LIN {X 0,Y 204.772,Z 618.344,A -85,B 0,C 180,E1 -29638.617,E2 -29638.617} C_VEL
LIN {X 0,Y 211.612,Z 616.813,A -85,B 0,C 180,E1 -29641.984,E2 -29641.984} C_VEL
LIN {X 0,Y 215.146,Z 615.633,A -85,B 0,C 180,E1 -29643.61,E2 -29643.61} C_VEL
LIN {X 0,Y 223.244,Z 612.344,A -85,B 0,C 180,E1 -29646.599,E2 -29646.599} C_VEL
LIN {X 0,Y 232.156,Z 607.768,A -85,B 0,C 180,E1 -29649.321,E2 -29649.321} C_VEL
LIN {X 0,Y 241.752,Z 601.799,A -85,B 0,C 180,E1 -29651.794,E2 -29651.794} C_VEL
LIN {X 0,Y 251.918,Z 594.305,A -85,B 0,C 180,E1 -29654.041,E2 -29654.041} C_VEL
LIN {X 0,Y 261.51,Z 586.109,A -85,B 0,C 180,E1 -29655.824,E2 -29655.824} C_VEL
LIN {X 0,Y 271.184,Z 576.576,A -85,B 0,C 180,E1 -29657.407,E2 -29657.407} C_VEL
LIN {X 0,Y 279.896,Z 566.683,A -85,B 0,C 180,E1 -29658.66,E2 -29658.66} C_VEL
LIN {X 0,Y 288.902,Z 554.834,A -85,B 0,C 180,E1 -29659.797,E2 -29659.797} C_VEL
LIN {X 0,Y 297.375,Z 541.679,A -85,B 0,C 180,E1 -29660.75,E2 -29660.75} C_VEL
LIN {X 0,Y 300.334,Z 536.479,A -85,B 0,C 180,E1 -29661.053,E2 -29661.053} C_VEL
LIN {X 0,Y 300.286,Z 536.529,A -85,B 0,C 180,E1 -29661.393,E2 -29661.393} C_VEL
LIN {X 0,Y 292.719,Z 549.042,A -85,B 0,C 180,E1 -29662.328,E2 -29662.328} C_VEL
LIN {X 0,Y 284.753,Z 560.194,A -85,B 0,C 180,E1 -29663.38,E2 -29663.38} C_VEL
LIN {X 0,Y 275.713,Z 571.006,A -85,B 0,C 180,E1 -29664.684,E2 -29664.684} C_VEL
LIN {X 0,Y 266.952,Z 580.103,A -85,B 0,C 180,E1 -29666.112,E2 -29666.112} C_VEL
LIN {X 0,Y 256.846,Z 589.123,A -85,B 0,C 180,E1 -29667.977,E2 -29667.977} C_VEL
LIN {X 0,Y 246.497,Z 596.964,A -85,B 0,C 180,E1 -29670.18,E2 -29670.18} C_VEL
LIN {X 0,Y 236.497,Z 603.258,A -85,B 0,C 180,E1 -29672.696,E2 -29672.696} C_VEL
LIN {X 0,Y 227.293,Z 607.968,A -85,B 0,C 180,E1 -29675.416,E2 -29675.416} C_VEL
LIN {X 0,Y 218.078,Z 611.557,A -85,B 0,C 180,E1 -29678.672,E2 -29678.672} C_VEL
LIN {X 0,Y 212.957,Z 613.013,A -85,B 0,C 180,E1 -29680.797,E2 -29680.797} C_VEL
LIN {X 0,Y 205.913,Z 614.151,A -85,B 0,C 180,E1 -29684.209,E2 -29684.209} C_VEL
LIN {X 0,Y 199.91,Z 614.063,A -85,B 0,C 180,E1 -29687.864,E2 -29687.864} C_VEL
LIN {X 0,Y 195.099,Z 612.779,A -85,B 0,C 180,E1 -29691.743,E2 -29691.743} C_VEL
LIN {X 0,Y 191.462,Z 610.312,A -85,B 0,C 180,E1 -29695.804,E2 -29695.804} C_VEL
LIN {X 0,Y 188.992,Z 606.632,A -85,B 0,C 180,E1 -29700,E2 -29700} C_VEL
LIN {X 0,Y 187.534,Z 601.624,A -85,B 0,C 180,E1 -29704.284,E2 -29704.284} C_VEL
LIN {X 0,Y 187.042,Z 595.113,A -85,B 0,C 180,E1 -29708.615,E2 -29708.615} C_VEL
LIN {X 0,Y 187.164,Z 587.88,A -85,B 0,C 180,E1 -29712.427,E2 -29712.427} C_VEL
LIN {X 0,Y 187.494,Z 580.247,A -85,B 0,C 180,E1 -29715.715,E2 -29715.715} C_VEL
LIN {X 0,Y 187.907,Z 570.867,A -85,B 0,C 180,E1 -29719.036,E2 -29719.036} C_VEL
LIN {X 0,Y 188.535,Z 560.39,A -85,B 0,C 180,E1 -29722.096,E2 -29722.096} C_VEL
LIN {X 0,Y 189.361,Z 548.884,A -85,B 0,C 180,E1 -29724.883,E2 -29724.883} C_VEL
LIN {X 0,Y 190.461,Z 535.611,A -85,B 0,C 180,E1 -29727.516,E2 -29727.516} C_VEL
LIN {X 0,Y 191.581,Z 521.627,A -85,B 0,C 180,E1 -29729.727,E2 -29729.727} C_VEL
LIN {X 0,Y 192.62,Z 507.163,A -85,B 0,C 180,E1 -29731.516,E2 -29731.516} C_VEL
LIN {X 0,Y 193.716,Z 492.08,A -85,B 0,C 180,E1 -29732.933,E2 -29732.933} C_VEL
LIN {X 0,Y 194.887,Z 470.161,A -85,B 0,C 180,E1 -29734.369,E2 -29734.369} C_VEL
LIN {X 0,Y 198.573,Z 392.946,A -85,B 0,C 180,E1 -29738.995,E2 -29738.995} C_VEL
LIN {X 0,Y 195.924,Z 362.092,A -85,B 0,C 180,E1 -29740.947,E2 -29740.947} C_VEL
LIN {X 0,Y 192.683,Z 347.917,A -85,B 0,C 180,E1 -29742.011,E2 -29742.011} C_VEL
LIN {X 0,Y 189.766,Z 333.395,A -85,B 0,C 180,E1 -29746.279,E2 -29746.279} C_VEL
LIN {X 0,Y 189.689,Z 333.409,A -85,B 0,C 180,E1 -29751.11,E2 -29751.11} C_VEL
LIN {X 0,Y 189.64,Z 333.393,A -85,B 0,C 180,E1 -29756.35,E2 -29756.35} C_VEL
LIN {X 0,Y 189.682,Z 333.399,A -85,B 0,C 180,E1 -29757.777,E2 -29757.777} C_VEL
LIN {X 0,Y 190.707,Z 336.248,A -85,B 0,C 180,E1 -29758.187,E2 -29758.187} C_VEL
LIN {X 0,Y 192.446,Z 338.584,A -85,B 0,C 180,E1 -29758.713,E2 -29758.713} C_VEL
LIN {X 0,Y 201.749,Z 354.151,A -85,B 0,C 180,E1 -29761.457,E2 -29761.457} C_VEL
LIN {X 0,Y 210.076,Z 370.517,A -85,B 0,C 180,E1 -29763.742,E2 -29763.742} C_VEL
LIN {X 0,Y 214.586,Z 381.294,A -85,B 0,C 180,E1 -29764.958,E2 -29764.958} C_VEL
LIN {X 0,Y 210.894,Z 456.713,A -85,B 0,C 180,E1 -29767.348,E2 -29767.348} C_VEL
LIN {X 0,Y 209.707,Z 470.555,A -85,B 0,C 180,E1 -29768.117,E2 -29768.117} C_VEL
LIN {X 0,Y 207.974,Z 484.658,A -85,B 0,C 180,E1 -29769.286,E2 -29769.286} C_VEL
LIN {X 0,Y 205.708,Z 498.601,A -85,B 0,C 180,E1 -29770.864,E2 -29770.864} C_VEL
LIN {X 0,Y 202.935,Z 511.157,A -85,B 0,C 180,E1 -29772.676,E2 -29772.676} C_VEL
LIN {X 0,Y 200.212,Z 522.577,A -85,B 0,C 180,E1 -29774.783,E2 -29774.783} C_VEL
LIN {X 0,Y 198.207,Z 531.077,A -85,B 0,C 180,E1 -29776.716,E2 -29776.716} C_VEL
LIN {X 0,Y 195.137,Z 541.849,A -85,B 0,C 180,E1 -29779.656,E2 -29779.656} C_VEL
LIN {X 0,Y 192.712,Z 550.717,A -85,B 0,C 180,E1 -29782.686,E2 -29782.686} C_VEL
LIN {X 0,Y 190.577,Z 558.125,A -85,B 0,C 180,E1 -29785.779,E2 -29785.779} C_VEL
LIN {X 0,Y 189.135,Z 564.829,A -85,B 0,C 180,E1 -29789.266,E2 -29789.266} C_VEL
LIN {X 0,Y 187.809,Z 570.83,A -85,B 0,C 180,E1 -29793.202,E2 -29793.202} C_VEL
LIN {X 0,Y 186.836,Z 575.79,A -85,B 0,C 180,E1 -29797.534,E2 -29797.534} C_VEL
LIN {X 0,Y 186.652,Z 578.504,A -85,B 0,C 180,E1 -29800.809,E2 -29800.809} C_VEL
LIN {X 0,Y 186.756,Z 579.872,A -85,B 0,C 180,E1 -29802.999,E2 -29802.999} C_VEL
LIN {X 0,Y 187.345,Z 581.595,A -85,B 0,C 180,E1 -29807.398,E2 -29807.398} C_VEL
LIN {X 0,Y 188.986,Z 581.937,A -85,B 0,C 180,E1 -29812.092,E2 -29812.092} C_VEL
LIN {X 0,Y 191.122,Z 580.952,A -85,B 0,C 180,E1 -29816.084,E2 -29816.084} C_VEL
LIN {X 0,Y 194.361,Z 578.551,A -85,B 0,C 180,E1 -29820.294,E2 -29820.294} C_VEL
LIN {X 0,Y 198.436,Z 574.642,A -85,B 0,C 180,E1 -29824.38,E2 -29824.38} C_VEL
LIN {X 0,Y 203.477,Z 569.082,A -85,B 0,C 180,E1 -29828.282,E2 -29828.282} C_VEL
LIN {X 0,Y 208.517,Z 562.735,A -85,B 0,C 180,E1 -29831.555,E2 -29831.555} C_VEL
LIN {X 0,Y 214.19,Z 554.762,A -85,B 0,C 180,E1 -29834.668,E2 -29834.668} C_VEL
LIN {X 0,Y 219.487,Z 546.356,A -85,B 0,C 180,E1 -29837.215,E2 -29837.215} C_VEL
LIN {X 0,Y 225.215,Z 536.161,A -85,B 0,C 180,E1 -29839.631,E2 -29839.631} C_VEL
LIN {X 0,Y 230.243,Z 525.826,A -85,B 0,C 180,E1 -29841.562,E2 -29841.562} C_VEL
LIN {X 0,Y 234.956,Z 514.4,A -85,B 0,C 180,E1 -29843.274,E2 -29843.274} C_VEL
LIN {X 0,Y 239.109,Z 502.35,A -85,B 0,C 180,E1 -29844.698,E2 -29844.698} C_VEL
LIN {X 0,Y 242.65,Z 489.425,A -85,B 0,C 180,E1 -29845.896,E2 -29845.896} C_VEL
LIN {X 0,Y 245.689,Z 475.198,A -85,B 0,C 180,E1 -29846.854,E2 -29846.854} C_VEL
LIN {X 0,Y 247.681,Z 461.5,A -85,B 0,C 180,E1 -29847.513,E2 -29847.513} C_VEL
LIN {X 0,Y 249.394,Z 440.592,A -85,B 0,C 180,E1 -29848.12,E2 -29848.12} C_VEL
LIN {X 0,Y 251.105,Z 416.237,A -85,B 0,C 180,E1 -29848.742,E2 -29848.742} C_VEL
LIN {X 0,Y 244.75,Z 404.193,A -85,B 0,C 180,E1 -29851.331,E2 -29851.331} C_VEL
LIN {X 0,Y 239.319,Z 395.049,A -85,B 0,C 180,E1 -29853.74,E2 -29853.74} C_VEL
LIN {X 0,Y 234.137,Z 386.937,A -85,B 0,C 180,E1 -29856.29,E2 -29856.29} C_VEL
LIN {X 0,Y 229.497,Z 380.171,A -85,B 0,C 180,E1 -29858.838,E2 -29858.838} C_VEL
LIN {X 0,Y 226.579,Z 376.111,A -85,B 0,C 180,E1 -29860.605,E2 -29860.605} C_VEL
LIN {X 0,Y 223.563,Z 371.946,A -85,B 0,C 180,E1 -29862.612,E2 -29862.612} C_VEL
LIN {X 0,Y 220.384,Z 367.707,A -85,B 0,C 180,E1 -29864.976,E2 -29864.976} C_VEL
LIN {X 0,Y 217.707,Z 364.529,A -85,B 0,C 180,E1 -29867.206,E2 -29867.206} C_VEL
LIN {X 0,Y 216.596,Z 362.722,A -85,B 0,C 180,E1 -29868.28,E2 -29868.28} C_VEL
LIN {X 0,Y 214.036,Z 360.136,A -85,B 0,C 180,E1 -29870.924,E2 -29870.924} C_VEL
LIN {X 0,Y 212.711,Z 357.426,A -85,B 0,C 180,E1 -29872.728,E2 -29872.728} C_VEL
LIN {X 0,Y 209.928,Z 355.08,A -85,B 0,C 180,E1 -29877.071,E2 -29877.071} C_VEL
LIN {X 0,Y 208.728,Z 352.105,A -85,B 0,C 180,E1 -29880.602,E2 -29880.602} C_VEL
LIN {X 0,Y 208.657,Z 351.751,A -85,B 0,C 180,E1 -29880.963,E2 -29880.963} C_VEL
LIN {X 0,Y 208.195,Z 351.882,A -85,B 0,C 180,E1 -29888.464,E2 -29888.464} C_VEL
LIN {X 0,Y 208.512,Z 352.77,A -85,B 0,C 180,E1 -29890.219,E2 -29890.219} C_VEL
LIN {X 0,Y 210.498,Z 356.559,A -85,B 0,C 180,E1 -29895.439,E2 -29895.439} C_VEL
LIN {X 0,Y 213.777,Z 361.036,A -85,B 0,C 180,E1 -29900.192,E2 -29900.192} C_VEL
LIN {X 0,Y 218.035,Z 367.529,A -85,B 0,C 180,E1 -29904.59,E2 -29904.59} C_VEL
LIN {X 0,Y 222.816,Z 375.197,A -85,B 0,C 180,E1 -29908.454,E2 -29908.454} C_VEL
LIN {X 0,Y 226.433,Z 381.12,A -85,B 0,C 180,E1 -29910.933,E2 -29910.933} C_VEL
LIN {X 0,Y 230.081,Z 387.521,A -85,B 0,C 180,E1 -29913.184,E2 -29913.184} C_VEL
LIN {X 0,Y 234.473,Z 395.589,A -85,B 0,C 180,E1 -29915.629,E2 -29915.629} C_VEL
LIN {X 0,Y 239.381,Z 405.545,A -85,B 0,C 180,E1 -29918.107,E2 -29918.107} C_VEL
LIN {X 0,Y 244.569,Z 417.022,A -85,B 0,C 180,E1 -29920.506,E2 -29920.506} C_VEL
LIN {X 0,Y 249.126,Z 428.767,A -85,B 0,C 180,E1 -29922.503,E2 -29922.503} C_VEL
LIN {X 0,Y 249.583,Z 430.837,A -85,B 0,C 180,E1 -29922.735,E2 -29922.735} C_VEL
LIN {X 0,Y 249.848,Z 436.032,A -85,B 0,C 180,E1 -29923.052,E2 -29923.052} C_VEL
LIN {X 0,Y 246.628,Z 477.617,A -85,B 0,C 180,E1 -29924.114,E2 -29924.114} C_VEL
LIN {X 0,Y 244.414,Z 491.839,A -85,B 0,C 180,E1 -29924.684,E2 -29924.684} C_VEL
LIN {X 0,Y 241.258,Z 506.122,A -85,B 0,C 180,E1 -29925.546,E2 -29925.546} C_VEL
LIN {X 0,Y 237.076,Z 519.77,A -85,B 0,C 180,E1 -29926.62,E2 -29926.62} C_VEL
LIN {X 0,Y 232.475,Z 532.04,A -85,B 0,C 180,E1 -29927.909,E2 -29927.909} C_VEL
LIN {X 0,Y 227.643,Z 543.281,A -85,B 0,C 180,E1 -29929.465,E2 -29929.465} C_VEL
LIN {X 0,Y 222.898,Z 552.692,A -85,B 0,C 180,E1 -29931.068,E2 -29931.068} C_VEL
LIN {X 0,Y 219.363,Z 559.338,A -85,B 0,C 180,E1 -29932.452,E2 -29932.452} C_VEL
LIN {X 0,Y 216.541,Z 563.417,A -85,B 0,C 180,E1 -29933.297,E2 -29933.297} C_VEL
LIN {X 0,Y 210.353,Z 569.669,A -85,B 0,C 180,E1 -29934.529,E2 -29934.529} C_VEL
LIN {X 0,Y 204.048,Z 575.426,A -85,B 0,C 180,E1 -29935.933,E2 -29935.933} C_VEL
LIN {X 0,Y 201.095,Z 578.671,A -85,B 0,C 180,E1 -29937.048,E2 -29937.048} C_VEL
LIN {X 0,Y 195.998,Z 585.222,A -85,B 0,C 180,E1 -29939.985,E2 -29939.985} C_VEL
LIN {X 0,Y 190.604,Z 591.683,A -85,B 0,C 180,E1 -29943.839,E2 -29943.839} C_VEL
LIN {X 0,Y 186.379,Z 596.566,A -85,B 0,C 180,E1 -29947.931,E2 -29947.931} C_VEL
LIN {X 0,Y 183.063,Z 600.003,A -85,B 0,C 180,E1 -29952.182,E2 -29952.182} C_VEL
LIN {X 0,Y 180.819,Z 602.091,A -85,B 0,C 180,E1 -29956.566,E2 -29956.566} C_VEL
LIN {X 0,Y 179.627,Z 602.882,A -85,B 0,C 180,E1 -29961.032,E2 -29961.032} C_VEL
LIN {X 0,Y 179.587,Z 602.391,A -85,B 0,C 180,E1 -29965.532,E2 -29965.532} C_VEL
LIN {X 0,Y 180.477,Z 600.589,A -85,B 0,C 180,E1 -29970.005,E2 -29970.005} C_VEL
LIN {X 0,Y 181.269,Z 598.812,A -85,B 0,C 180,E1 -29972.774,E2 -29972.774} C_VEL
LIN {X 0,Y 180.846,Z 604.623,A -85,B 0,C 180,E1 -29976.678,E2 -29976.678} C_VEL
LIN {X 0,Y 181.12,Z 609.795,A -85,B 0,C 180,E1 -29981.154,E2 -29981.154} C_VEL
LIN {X 0,Y 182.865,Z 613.729,A -85,B 0,C 180,E1 -29985.558,E2 -29985.558} C_VEL
LIN {X 0,Y 185.901,Z 616.471,A -85,B 0,C 180,E1 -29989.828,E2 -29989.828} C_VEL
LIN {X 0,Y 190.04,Z 618.055,A -85,B 0,C 180,E1 -29993.924,E2 -29993.924} C_VEL
LIN {X 0,Y 195.425,Z 618.533,A -85,B 0,C 180,E1 -29997.777,E2 -29997.777} C_VEL
LIN {X 0,Y 202.009,Z 617.902,A -85,B 0,C 180,E1 -30001.345,E2 -30001.345} C_VEL
LIN {X 0,Y 209.302,Z 616.159,A -85,B 0,C 180,E1 -30004.68,E2 -30004.68} C_VEL
LIN {X 0,Y 217.637,Z 613.252,A -85,B 0,C 180,E1 -30007.703,E2 -30007.703} C_VEL
LIN {X 0,Y 226.788,Z 609.104,A -85,B 0,C 180,E1 -30010.441,E2 -30010.441} C_VEL
LIN {X 0,Y 236.63,Z 603.619,A -85,B 0,C 180,E1 -30012.913,E2 -30012.913} C_VEL
LIN {X 0,Y 247.027,Z 596.699,A -85,B 0,C 180,E1 -30015.148,E2 -30015.148} C_VEL
LIN {X 0,Y 255.69,Z 590.016,A -85,B 0,C 180,E1 -30016.73,E2 -30016.73} C_VEL
LIN {X 0,Y 265.231,Z 581.579,A -85,B 0,C 180,E1 -30018.254,E2 -30018.254} C_VEL
LIN {X 0,Y 274.014,Z 572.664,A -85,B 0,C 180,E1 -30019.511,E2 -30019.511} C_VEL
LIN {X 0,Y 283.084,Z 562.119,A -85,B 0,C 180,E1 -30020.649,E2 -30020.649} C_VEL
LIN {X 0,Y 287.744,Z 556.036,A -85,B 0,C 180,E1 -30021.17,E2 -30021.17} C_VEL
LIN {X 0,Y 287.155,Z 556.784,A -85,B 0,C 180,E1 -30021.519,E2 -30021.519} C_VEL
LIN {X 0,Y 277.723,Z 568.304,A -85,B 0,C 180,E1 -30022.749,E2 -30022.749} C_VEL
LIN {X 0,Y 268.759,Z 577.696,A -85,B 0,C 180,E1 -30024.037,E2 -30024.037} C_VEL
LIN {X 0,Y 258.34,Z 587.079,A -85,B 0,C 180,E1 -30025.764,E2 -30025.764} C_VEL
LIN {X 0,Y 248.476,Z 594.599,A -85,B 0,C 180,E1 -30027.615,E2 -30027.615} C_VEL
LIN {X 0,Y 240.38,Z 599.92,A -85,B 0,C 180,E1 -30029.341,E2 -30029.341} C_VEL
LIN {X 0,Y 230.458,Z 605.455,A -85,B 0,C 180,E1 -30031.82,E2 -30031.82} C_VEL
LIN {X 0,Y 223.097,Z 608.777,A -85,B 0,C 180,E1 -30033.925,E2 -30033.925} C_VEL
LIN {X 0,Y 214.2,Z 611.931,A -85,B 0,C 180,E1 -30036.896,E2 -30036.896} C_VEL
LIN {X 0,Y 206.151,Z 613.805,A -85,B 0,C 180,E1 -30040.137,E2 -30040.137} C_VEL
LIN {X 0,Y 198.965,Z 614.461,A -85,B 0,C 180,E1 -30043.642,E2 -30043.642} C_VEL
LIN {X 0,Y 192.894,Z 613.909,A -85,B 0,C 180,E1 -30047.416,E2 -30047.416} C_VEL
LIN {X 0,Y 188.015,Z 612.183,A -85,B 0,C 180,E1 -30051.43,E2 -30051.43} C_VEL
LIN {X 0,Y 184.356,Z 609.288,A -85,B 0,C 180,E1 -30055.642,E2 -30055.642} C_VEL
LIN {X 0,Y 181.653,Z 604.435,A -85,B 0,C 180,E1 -30060.679,E2 -30060.679} C_VEL
LIN {X 0,Y 180.539,Z 599.69,A -85,B 0,C 180,E1 -30064.45,E2 -30064.45} C_VEL
LIN {X 0,Y 180.131,Z 592.661,A -85,B 0,C 180,E1 -30068.948,E2 -30068.948} C_VEL
LIN {X 0,Y 180.336,Z 584.928,A -85,B 0,C 180,E1 -30072.905,E2 -30072.905} C_VEL
LIN {X 0,Y 180.656,Z 576.677,A -85,B 0,C 180,E1 -30076.326,E2 -30076.326} C_VEL
LIN {X 0,Y 181.143,Z 566.602,A -85,B 0,C 180,E1 -30079.776,E2 -30079.776} C_VEL
LIN {X 0,Y 181.822,Z 555.241,A -85,B 0,C 180,E1 -30082.958,E2 -30082.958} C_VEL
LIN {X 0,Y 182.745,Z 542.615,A -85,B 0,C 180,E1 -30085.849,E2 -30085.849} C_VEL
LIN {X 0,Y 183.856,Z 529.323,A -85,B 0,C 180,E1 -30088.332,E2 -30088.332} C_VEL
LIN {X 0,Y 185.016,Z 515.203,A -85,B 0,C 180,E1 -30090.422,E2 -30090.422} C_VEL
LIN {X 0,Y 186.085,Z 500.378,A -85,B 0,C 180,E1 -30092.119,E2 -30092.119} C_VEL
LIN {X 0,Y 187.091,Z 484.465,A -85,B 0,C 180,E1 -30093.439,E2 -30093.439} C_VEL
LIN {X 0,Y 191.458,Z 393.062,A -85,B 0,C 180,E1 -30099.202,E2 -30099.202} C_VEL
LIN {X 0,Y 188.969,Z 363.416,A -85,B 0,C 180,E1 -30101.142,E2 -30101.142} C_VEL
LIN {X 0,Y 185.562,Z 348.298,A -85,B 0,C 180,E1 -30102.257,E2 -30102.257} C_VEL
LIN {X 0,Y 182.722,Z 334.274,A -85,B 0,C 180,E1 -30106.511,E2 -30106.511} C_VEL
LIN {X 0,Y 182.589,Z 334.299,A -85,B 0,C 180,E1 -30112.13,E2 -30112.13} C_VEL
LIN {X 0,Y 182.589,Z 334.283,A -85,B 0,C 180,E1 -30116,E2 -30116} C_VEL
LIN {X 0,Y 183.502,Z 336.96,A -85,B 0,C 180,E1 -30116.385,E2 -30116.385} C_VEL
LIN {X 0,Y 185.484,Z 339.565,A -85,B 0,C 180,E1 -30117.04,E2 -30117.04} C_VEL
LIN {X 0,Y 192.367,Z 350.608,A -85,B 0,C 180,E1 -30119.258,E2 -30119.258} C_VEL
LIN {X 0,Y 199.468,Z 363.339,A -85,B 0,C 180,E1 -30121.389,E2 -30121.389} C_VEL
LIN {X 0,Y 206.415,Z 377.842,A -85,B 0,C 180,E1 -30123.371,E2 -30123.371} C_VEL
LIN {X 0,Y 208.518,Z 383.493,A -85,B 0,C 180,E1 -30123.989,E2 -30123.989} C_VEL
LIN {X 0,Y 204.686,Z 458.09,A -85,B 0,C 180,E1 -30126.42,E2 -30126.42} C_VEL
LIN {X 0,Y 203.379,Z 472.341,A -85,B 0,C 180,E1 -30127.266,E2 -30127.266} C_VEL
LIN {X 0,Y 201.579,Z 486.089,A -85,B 0,C 180,E1 -30128.463,E2 -30128.463} C_VEL
LIN {X 0,Y 199.383,Z 498.938,A -85,B 0,C 180,E1 -30129.964,E2 -30129.964} C_VEL
LIN {X 0,Y 196.504,Z 511.51,A -85,B 0,C 180,E1 -30131.822,E2 -30131.822} C_VEL
LIN {X 0,Y 193.678,Z 522.939,A -85,B 0,C 180,E1 -30133.988,E2 -30133.988} C_VEL
LIN {X 0,Y 191.291,Z 532.424,A -85,B 0,C 180,E1 -30136.226,E2 -30136.226} C_VEL
LIN {X 0,Y 188.155,Z 543.039,A -85,B 0,C 180,E1 -30139.268,E2 -30139.268} C_VEL
LIN {X 0,Y 185.679,Z 551.775,A -85,B 0,C 180,E1 -30142.408,E2 -30142.408} C_VEL
LIN {X 0,Y 183.513,Z 559.068,A -85,B 0,C 180,E1 -30145.617,E2 -30145.617} C_VEL
LIN {X 0,Y 182.15,Z 565.101,A -85,B 0,C 180,E1 -30148.888,E2 -30148.888} C_VEL
LIN {X 0,Y 180.98,Z 570.15,A -85,B 0,C 180,E1 -30152.213,E2 -30152.213} C_VEL
LIN {X 0,Y 179.846,Z 575.381,A -85,B 0,C 180,E1 -30156.704,E2 -30156.704} C_VEL
LIN {X 0,Y 179.581,Z 579.098,A -85,B 0,C 180,E1 -30161.24,E2 -30161.24} C_VEL
LIN {X 0,Y 179.935,Z 581.425,A -85,B 0,C 180,E1 -30165.807,E2 -30165.807} C_VEL
LIN {X 0,Y 181.136,Z 582.388,A -85,B 0,C 180,E1 -30170.36,E2 -30170.36} C_VEL
LIN {X 0,Y 183.213,Z 581.991,A -85,B 0,C 180,E1 -30174.863,E2 -30174.863} C_VEL
LIN {X 0,Y 186.2,Z 580.215,A -85,B 0,C 180,E1 -30179.27,E2 -30179.27} C_VEL
LIN {X 0,Y 190.117,Z 576.967,A -85,B 0,C 180,E1 -30183.542,E2 -30183.542} C_VEL
LIN {X 0,Y 194.975,Z 572.149,A -85,B 0,C 180,E1 -30187.635,E2 -30187.635} C_VEL
LIN {X 0,Y 199.221,Z 567.445,A -85,B 0,C 180,E1 -30190.568,E2 -30190.568} C_VEL
LIN {X 0,Y 205.163,Z 559.989,A -85,B 0,C 180,E1 -30194.061,E2 -30194.061} C_VEL
LIN {X 0,Y 210.85,Z 551.891,A -85,B 0,C 180,E1 -30196.949,E2 -30196.949} C_VEL
LIN {X 0,Y 216.113,Z 543.516,A -85,B 0,C 180,E1 -30199.289,E2 -30199.289} C_VEL
LIN {X 0,Y 221.568,Z 533.678,A -85,B 0,C 180,E1 -30201.475,E2 -30201.475} C_VEL
LIN {X 0,Y 226.813,Z 522.733,A -85,B 0,C 180,E1 -30203.402,E2 -30203.402} C_VEL
LIN {X 0,Y 231.709,Z 510.682,A -85,B 0,C 180,E1 -30205.074,E2 -30205.074} C_VEL
LIN {X 0,Y 236.126,Z 497.237,A -85,B 0,C 180,E1 -30206.534,E2 -30206.534} C_VEL
LIN {X 0,Y 239.487,Z 484.106,A -85,B 0,C 180,E1 -30207.612,E2 -30207.612} C_VEL
LIN {X 0,Y 242.123,Z 470.077,A -85,B 0,C 180,E1 -30208.457,E2 -30208.457} C_VEL
LIN {X 0,Y 243.851,Z 456.722,A -85,B 0,C 180,E1 -30208.986,E2 -30208.986} C_VEL
LIN {X 0,Y 246.627,Z 419.248,A -85,B 0,C 180,E1 -30209.972,E2 -30209.972} C_VEL
LIN {X 0,Y 240.564,Z 407.702,A -85,B 0,C 180,E1 -30212.598,E2 -30212.598} C_VEL
LIN {X 0,Y 234.866,Z 397.966,A -85,B 0,C 180,E1 -30215.322,E2 -30215.322} C_VEL
LIN {X 0,Y 229.142,Z 389.098,A -85,B 0,C 180,E1 -30218.409,E2 -30218.409} C_VEL
LIN {X 0,Y 224.548,Z 382.445,A -85,B 0,C 180,E1 -30221.235,E2 -30221.235} C_VEL
LIN {X 0,Y 221.699,Z 378.424,A -85,B 0,C 180,E1 -30223.209,E2 -30223.209} C_VEL
LIN {X 0,Y 218.549,Z 374.165,A -85,B 0,C 180,E1 -30225.651,E2 -30225.651} C_VEL
LIN {X 0,Y 215.838,Z 370.597,A -85,B 0,C 180,E1 -30228.06,E2 -30228.06} C_VEL
LIN {X 0,Y 215.173,Z 369.487,A -85,B 0,C 180,E1 -30228.737,E2 -30228.737} C_VEL
LIN {X 0,Y 212.724,Z 366.921,A -85,B 0,C 180,E1 -30231.382,E2 -30231.382} C_VEL
LIN {X 0,Y 211.388,Z 364.233,A -85,B 0,C 180,E1 -30233.281,E2 -30233.281} C_VEL
LIN {X 0,Y 208.826,Z 361.893,A -85,B 0,C 180,E1 -30237.537,E2 -30237.537} C_VEL
LIN {X 0,Y 207.733,Z 358.915,A -85,B 0,C 180,E1 -30241.088,E2 -30241.088} C_VEL
LIN {X 0,Y 207.277,Z 358.832,A -85,B 0,C 180,E1 -30248.135,E2 -30248.135} C_VEL
LIN {X 0,Y 207.592,Z 359.88,A -85,B 0,C 180,E1 -30250.081,E2 -30250.081} C_VEL
LIN {X 0,Y 209.354,Z 363.349,A -85,B 0,C 180,E1 -30254.968,E2 -30254.968} C_VEL
LIN {X 0,Y 212.393,Z 367.71,A -85,B 0,C 180,E1 -30259.632,E2 -30259.632} C_VEL
LIN {X 0,Y 216.794,Z 374.826,A -85,B 0,C 180,E1 -30264.375,E2 -30264.375} C_VEL
LIN {X 0,Y 220.837,Z 381.482,A -85,B 0,C 180,E1 -30267.76,E2 -30267.76} C_VEL
LIN {X 0,Y 224.206,Z 387.201,A -85,B 0,C 180,E1 -30270.185,E2 -30270.185} C_VEL
LIN {X 0,Y 227.691,Z 393.527,A -85,B 0,C 180,E1 -30272.441,E2 -30272.441} C_VEL
LIN {X 0,Y 231.925,Z 401.659,A -85,B 0,C 180,E1 -30274.916,E2 -30274.916} C_VEL
LIN {X 0,Y 236.147,Z 410.507,A -85,B 0,C 180,E1 -30277.165,E2 -30277.165} C_VEL
LIN {X 0,Y 241.32,Z 422.337,A -85,B 0,C 180,E1 -30279.685,E2 -30279.685} C_VEL
LIN {X 0,Y 245.219,Z 432.773,A -85,B 0,C 180,E1 -30281.492,E2 -30281.492} C_VEL
LIN {X 0,Y 245.473,Z 436.81,A -85,B 0,C 180,E1 -30281.768,E2 -30281.768} C_VEL
LIN {X 0,Y 242.262,Z 477.025,A -85,B 0,C 180,E1 -30282.796,E2 -30282.796} C_VEL
LIN {X 0,Y 239.971,Z 491.43,A -85,B 0,C 180,E1 -30283.373,E2 -30283.373} C_VEL
LIN {X 0,Y 236.872,Z 505.146,A -85,B 0,C 180,E1 -30284.192,E2 -30284.192} C_VEL
LIN {X 0,Y 232.593,Z 518.909,A -85,B 0,C 180,E1 -30285.264,E2 -30285.264} C_VEL
LIN {X 0,Y 227.867,Z 531.26,A -85,B 0,C 180,E1 -30286.551,E2 -30286.551} C_VEL
LIN {X 0,Y 222.314,Z 543.732,A -85,B 0,C 180,E1 -30288.28,E2 -30288.28} C_VEL
LIN {X 0,Y 216.413,Z 554.897,A -85,B 0,C 180,E1 -30290.272,E2 -30290.272} C_VEL
LIN {X 0,Y 210.553,Z 564.93,A -85,B 0,C 180,E1 -30292.625,E2 -30292.625} C_VEL
LIN {X 0,Y 205,Z 573.287,A -85,B 0,C 180,E1 -30295.088,E2 -30295.088} C_VEL
LIN {X 0,Y 201.095,Z 578.671,A -85,B 0,C 180,E1 -30297.048,E2 -30297.048} C_VEL
LIN {X 0,Y 198.172,Z 581.765,A -85,B 0,C 180,E1 -30298.233,E2 -30298.233} C_VEL
LIN {X 0,Y 191.953,Z 586.359,A -85,B 0,C 180,E1 -30300.068,E2 -30300.068} C_VEL
LIN {X 0,Y 185.92,Z 590.363,A -85,B 0,C 180,E1 -30302.116,E2 -30302.116} C_VEL
LIN {X 0,Y 183.346,Z 592.505,A -85,B 0,C 180,E1 -30303.617,E2 -30303.617} C_VEL
LIN {X 0,Y 179.772,Z 596.346,A -85,B 0,C 180,E1 -30307.075,E2 -30307.075} C_VEL
LIN {X 0,Y 176.276,Z 599.709,A -85,B 0,C 180,E1 -30311.471,E2 -30311.471} C_VEL
LIN {X 0,Y 173.892,Z 601.729,A -85,B 0,C 180,E1 -30316.02,E2 -30316.02} C_VEL
LIN {X 0,Y 172.597,Z 602.455,A -85,B 0,C 180,E1 -30320.664,E2 -30320.664} C_VEL
LIN {X 0,Y 172.487,Z 601.902,A -85,B 0,C 180,E1 -30325.347,E2 -30325.347} C_VEL
LIN {X 0,Y 173.395,Z 600.041,A -85,B 0,C 180,E1 -30330.006,E2 -30330.006} C_VEL
LIN {X 0,Y 174.408,Z 597.861,A -85,B 0,C 180,E1 -30333.531,E2 -30333.531} C_VEL
LIN {X 0,Y 174.002,Z 604.357,A -85,B 0,C 180,E1 -30338.105,E2 -30338.105} C_VEL
LIN {X 0,Y 174.672,Z 609.51,A -85,B 0,C 180,E1 -30342.747,E2 -30342.747} C_VEL
LIN {X 0,Y 176.127,Z 612.532,A -85,B 0,C 180,E1 -30346.169,E2 -30346.169} C_VEL
LIN {X 0,Y 179.304,Z 615.567,A -85,B 0,C 180,E1 -30350.59,E2 -30350.59} C_VEL
LIN {X 0,Y 183.596,Z 617.465,A -85,B 0,C 180,E1 -30354.819,E2 -30354.819} C_VEL
LIN {X 0,Y 189.185,Z 618.289,A -85,B 0,C 180,E1 -30358.777,E2 -30358.777} C_VEL
LIN {X 0,Y 195.988,Z 618.019,A -85,B 0,C 180,E1 -30362.423,E2 -30362.423} C_VEL
LIN {X 0,Y 203.539,Z 616.632,A -85,B 0,C 180,E1 -30365.81,E2 -30365.81} C_VEL
LIN {X 0,Y 212.116,Z 614.103,A -85,B 0,C 180,E1 -30368.865,E2 -30368.865} C_VEL
LIN {X 0,Y 221.494,Z 610.385,A -85,B 0,C 180,E1 -30371.618,E2 -30371.618} C_VEL
LIN {X 0,Y 231.594,Z 605.377,A -85,B 0,C 180,E1 -30374.082,E2 -30374.082} C_VEL
LIN {X 0,Y 242.221,Z 598.994,A -85,B 0,C 180,E1 -30376.303,E2 -30376.303} C_VEL
LIN {X 0,Y 253.464,Z 590.94,A -85,B 0,C 180,E1 -30378.262,E2 -30378.262} C_VEL
LIN {X 0,Y 263.733,Z 582.31,A -85,B 0,C 180,E1 -30379.784,E2 -30379.784} C_VEL
LIN {X 0,Y 272.911,Z 573.432,A -85,B 0,C 180,E1 -30381.009,E2 -30381.009} C_VEL
LIN {X 0,Y 274.253,Z 572.015,A -85,B 0,C 180,E1 -30381.171,E2 -30381.171} C_VEL
LIN {X 0,Y 275.082,Z 571.122,A -85,B 0,C 180,E1 -30381.494,E2 -30381.494} C_VEL
LIN {X 0,Y 266.013,Z 579.997,A -85,B 0,C 180,E1 -30382.727,E2 -30382.727} C_VEL
LIN {X 0,Y 255.493,Z 588.824,A -85,B 0,C 180,E1 -30384.368,E2 -30384.368} C_VEL
LIN {X 0,Y 245.149,Z 596.187,A -85,B 0,C 180,E1 -30386.203,E2 -30386.203} C_VEL
LIN {X 0,Y 234.305,Z 602.646,A -85,B 0,C 180,E1 -30388.456,E2 -30388.456} C_VEL
LIN {X 0,Y 224.641,Z 607.341,A -85,B 0,C 180,E1 -30390.823,E2 -30390.823} C_VEL
LIN {X 0,Y 216.671,Z 610.445,A -85,B 0,C 180,E1 -30393.09,E2 -30393.09} C_VEL
LIN {X 0,Y 207.569,Z 613.063,A -85,B 0,C 180,E1 -30396.112,E2 -30396.112} C_VEL
LIN {X 0,Y 199.363,Z 614.432,A -85,B 0,C 180,E1 -30399.43,E2 -30399.43} C_VEL
LIN {X 0,Y 192.034,Z 614.602,A -85,B 0,C 180,E1 -30403.034,E2 -30403.034} C_VEL
LIN {X 0,Y 185.879,Z 613.591,A -85,B 0,C 180,E1 -30406.933,E2 -30406.933} C_VEL
LIN {X 0,Y 180.952,Z 611.426,A -85,B 0,C 180,E1 -30411.093,E2 -30411.093} C_VEL
LIN {X 0,Y 177.28,Z 608.091,A -85,B 0,C 180,E1 -30415.468,E2 -30415.468} C_VEL
LIN {X 0,Y 174.744,Z 603.067,A -85,B 0,C 180,E1 -30420.396,E2 -30420.396} C_VEL
LIN {X 0,Y 173.576,Z 597.579,A -85,B 0,C 180,E1 -30424.629,E2 -30424.629} C_VEL
LIN {X 0,Y 173.279,Z 590.015,A -85,B 0,C 180,E1 -30429.305,E2 -30429.305} C_VEL
LIN {X 0,Y 173.517,Z 581.675,A -85,B 0,C 180,E1 -30433.421,E2 -30433.421} C_VEL
LIN {X 0,Y 173.861,Z 572.811,A -85,B 0,C 180,E1 -30436.983,E2 -30436.983} C_VEL
LIN {X 0,Y 174.315,Z 563.879,A -85,B 0,C 180,E1 -30439.971,E2 -30439.971} C_VEL
LIN {X 0,Y 175.003,Z 552.107,A -85,B 0,C 180,E1 -30443.251,E2 -30443.251} C_VEL
LIN {X 0,Y 175.871,Z 540.18,A -85,B 0,C 180,E1 -30445.983,E2 -30445.983} C_VEL
LIN {X 0,Y 176.918,Z 527.451,A -85,B 0,C 180,E1 -30448.366,E2 -30448.366} C_VEL
LIN {X 0,Y 178.086,Z 512.604,A -85,B 0,C 180,E1 -30450.569,E2 -30450.569} C_VEL
LIN {X 0,Y 179.177,Z 497.624,A -85,B 0,C 180,E1 -30452.266,E2 -30452.266} C_VEL
LIN {X 0,Y 180.209,Z 480.632,A -85,B 0,C 180,E1 -30453.633,E2 -30453.633} C_VEL
LIN {X 0,Y 184.383,Z 393.363,A -85,B 0,C 180,E1 -30459.384,E2 -30459.384} C_VEL
LIN {X 0,Y 181.966,Z 364.608,A -85,B 0,C 180,E1 -30461.347,E2 -30461.347} C_VEL
LIN {X 0,Y 178.291,Z 348.149,A -85,B 0,C 180,E1 -30462.652,E2 -30462.652} C_VEL
LIN {X 0,Y 175.649,Z 335.156,A -85,B 0,C 180,E1 -30466.737,E2 -30466.737} C_VEL
LIN {X 0,Y 175.548,Z 335.167,A -85,B 0,C 180,E1 -30470.321,E2 -30470.321} C_VEL
LIN {X 0,Y 175.567,Z 335.238,A -85,B 0,C 180,E1 -30474.024,E2 -30474.024} C_VEL
LIN {X 0,Y 176.549,Z 337.97,A -85,B 0,C 180,E1 -30474.471,E2 -30474.471} C_VEL
LIN {X 0,Y 178.567,Z 340.559,A -85,B 0,C 180,E1 -30475.202,E2 -30475.202} C_VEL
LIN {X 0,Y 180.771,Z 343.871,A -85,B 0,C 180,E1 -30475.998,E2 -30475.998} C_VEL
LIN {X 0,Y 187.791,Z 355.245,A -85,B 0,C 180,E1 -30478.391,E2 -30478.391} C_VEL
LIN {X 0,Y 194.202,Z 366.862,A -85,B 0,C 180,E1 -30480.422,E2 -30480.422} C_VEL
LIN {X 0,Y 201.048,Z 381.266,A -85,B 0,C 180,E1 -30482.486,E2 -30482.486} C_VEL
LIN {X 0,Y 202.45,Z 384.678,A -85,B 0,C 180,E1 -30482.906,E2 -30482.906} C_VEL
LIN {X 0,Y 198.72,Z 457.1,A -85,B 0,C 180,E1 -30485.32,E2 -30485.32} C_VEL
LIN {X 0,Y 197.462,Z 471.111,A -85,B 0,C 180,E1 -30486.128,E2 -30486.128} C_VEL
LIN {X 0,Y 195.579,Z 485.285,A -85,B 0,C 180,E1 -30487.351,E2 -30487.351} C_VEL
LIN {X 0,Y 193.489,Z 497.512,A -85,B 0,C 180,E1 -30488.771,E2 -30488.771} C_VEL
LIN {X 0,Y 190.51,Z 510.429,A -85,B 0,C 180,E1 -30490.671,E2 -30490.671} C_VEL
LIN {X 0,Y 187.539,Z 522.121,A -85,B 0,C 180,E1 -30492.89,E2 -30492.89} C_VEL
LIN {X 0,Y 184.987,Z 531.819,A -85,B 0,C 180,E1 -30495.187,E2 -30495.187} C_VEL
LIN {X 0,Y 181.673,Z 542.604,A -85,B 0,C 180,E1 -30498.316,E2 -30498.316} C_VEL
LIN {X 0,Y 179.038,Z 551.483,A -85,B 0,C 180,E1 -30501.558,E2 -30501.558} C_VEL
LIN {X 0,Y 176.724,Z 558.901,A -85,B 0,C 180,E1 -30504.878,E2 -30504.878} C_VEL
LIN {X 0,Y 175.033,Z 565.954,A -85,B 0,C 180,E1 -30508.847,E2 -30508.847} C_VEL
LIN {X 0,Y 173.844,Z 570.907,A -85,B 0,C 180,E1 -30512.303,E2 -30512.303} C_VEL
LIN {X 0,Y 172.701,Z 576.056,A -85,B 0,C 180,E1 -30516.983,E2 -30516.983} C_VEL
LIN {X 0,Y 172.523,Z 579.693,A -85,B 0,C 180,E1 -30521.706,E2 -30521.706} C_VEL
LIN {X 0,Y 172.939,Z 581.947,A -85,B 0,C 180,E1 -30526.464,E2 -30526.464} C_VEL
LIN {X 0,Y 174.309,Z 582.832,A -85,B 0,C 180,E1 -30531.196,E2 -30531.196} C_VEL
LIN {X 0,Y 176.595,Z 582.356,A -85,B 0,C 180,E1 -30535.862,E2 -30535.862} C_VEL
LIN {X 0,Y 179.84,Z 580.474,A -85,B 0,C 180,E1 -30540.413,E2 -30540.413} C_VEL
LIN {X 0,Y 184.041,Z 577.131,A -85,B 0,C 180,E1 -30544.805,E2 -30544.805} C_VEL
LIN {X 0,Y 189.238,Z 572.224,A -85,B 0,C 180,E1 -30548.987,E2 -30548.987} C_VEL
LIN {X 0,Y 193.695,Z 567.425,A -85,B 0,C 180,E1 -30551.982,E2 -30551.982} C_VEL
LIN {X 0,Y 199.941,Z 559.878,A -85,B 0,C 180,E1 -30555.521,E2 -30555.521} C_VEL
LIN {X 0,Y 205.917,Z 551.658,A -85,B 0,C 180,E1 -30558.439,E2 -30558.439} C_VEL
LIN {X 0,Y 211.851,Z 542.454,A -85,B 0,C 180,E1 -30560.965,E2 -30560.965} C_VEL
LIN {X 0,Y 217.625,Z 532.168,A -85,B 0,C 180,E1 -30563.181,E2 -30563.181} C_VEL
LIN {X 0,Y 222.52,Z 522.023,A -85,B 0,C 180,E1 -30564.918,E2 -30564.918} C_VEL
LIN {X 0,Y 227.588,Z 509.721,A -85,B 0,C 180,E1 -30566.588,E2 -30566.588} C_VEL
LIN {X 0,Y 231.89,Z 496.782,A -85,B 0,C 180,E1 -30567.948,E2 -30567.948} C_VEL
LIN {X 0,Y 235.052,Z 484.684,A -85,B 0,C 180,E1 -30568.942,E2 -30568.942} C_VEL
LIN {X 0,Y 237.753,Z 470.851,A -85,B 0,C 180,E1 -30569.781,E2 -30569.781} C_VEL
LIN {X 0,Y 239.542,Z 457.615,A -85,B 0,C 180,E1 -30570.312,E2 -30570.312} C_VEL
LIN {X 0,Y 242.25,Z 422.317,A -85,B 0,C 180,E1 -30571.25,E2 -30571.25} C_VEL
LIN {X 0,Y 236.099,Z 410.467,A -85,B 0,C 180,E1 -30574.105,E2 -30574.105} C_VEL
LIN {X 0,Y 229.922,Z 400.04,A -85,B 0,C 180,E1 -30577.329,E2 -30577.329} C_VEL
LIN {X 0,Y 225.048,Z 392.492,A -85,B 0,C 180,E1 -30580.223,E2 -30580.223} C_VEL
LIN {X 0,Y 221.956,Z 387.973,A -85,B 0,C 180,E1 -30582.282,E2 -30582.282} C_VEL
LIN {X 0,Y 219.551,Z 384.477,A -85,B 0,C 180,E1 -30584.05,E2 -30584.05} C_VEL
LIN {X 0,Y 216.891,Z 380.742,A -85,B 0,C 180,E1 -30586.219,E2 -30586.219} C_VEL
LIN {X 0,Y 214.241,Z 377.114,A -85,B 0,C 180,E1 -30588.687,E2 -30588.687} C_VEL
LIN {X 0,Y 213.62,Z 376.164,A -85,B 0,C 180,E1 -30589.349,E2 -30589.349} C_VEL
LIN {X 0,Y 211.233,Z 373.341,A -85,B 0,C 180,E1 -30592.108,E2 -30592.108} C_VEL
LIN {X 0,Y 210.121,Z 371.076,A -85,B 0,C 180,E1 -30593.78,E2 -30593.78} C_VEL
LIN {X 0,Y 207.709,Z 368.674,A -85,B 0,C 180,E1 -30598.068,E2 -30598.068} C_VEL
LIN {X 0,Y 206.746,Z 365.792,A -85,B 0,C 180,E1 -30601.578,E2 -30601.578} C_VEL
LIN {X 0,Y 206.407,Z 365.932,A -85,B 0,C 180,E1 -30608.17,E2 -30608.17} C_VEL
LIN {X 0,Y 206.72,Z 367.122,A -85,B 0,C 180,E1 -30610.161,E2 -30610.161} C_VEL
LIN {X 0,Y 208.402,Z 370.502,A -85,B 0,C 180,E1 -30614.874,E2 -30614.874} C_VEL
LIN {X 0,Y 211.092,Z 374.505,A -85,B 0,C 180,E1 -30619.156,E2 -30619.156} C_VEL
LIN {X 0,Y 215.262,Z 381.576,A -85,B 0,C 180,E1 -30623.873,E2 -30623.873} C_VEL
LIN {X 0,Y 218.9,Z 387.798,A -85,B 0,C 180,E1 -30627.064,E2 -30627.064} C_VEL
LIN {X 0,Y 222.177,Z 393.587,A -85,B 0,C 180,E1 -30629.536,E2 -30629.536} C_VEL
LIN {X 0,Y 225.426,Z 399.704,A -85,B 0,C 180,E1 -30631.739,E2 -30631.739} C_VEL
LIN {X 0,Y 229.859,Z 408.661,A -85,B 0,C 180,E1 -30634.446,E2 -30634.446} C_VEL
LIN {X 0,Y 234.145,Z 418.078,A -85,B 0,C 180,E1 -30636.815,E2 -30636.815} C_VEL
LIN {X 0,Y 238.479,Z 428.666,A -85,B 0,C 180,E1 -30639.024,E2 -30639.024} C_VEL
LIN {X 0,Y 241.161,Z 436.292,A -85,B 0,C 180,E1 -30640.347,E2 -30640.347} C_VEL
LIN {X 0,Y 241.021,Z 440.551,A -85,B 0,C 180,E1 -30640.517,E2 -30640.517} C_VEL
LIN {X 0,Y 237.971,Z 476.878,A -85,B 0,C 180,E1 -30641.444,E2 -30641.444} C_VEL
LIN {X 0,Y 235.656,Z 491.06,A -85,B 0,C 180,E1 -30642.013,E2 -30642.013} C_VEL
LIN {X 0,Y 232.326,Z 505.322,A -85,B 0,C 180,E1 -30642.868,E2 -30642.868} C_VEL
LIN {X 0,Y 228.236,Z 518.08,A -85,B 0,C 180,E1 -30643.853,E2 -30643.853} C_VEL
LIN {X 0,Y 223.389,Z 530.508,A -85,B 0,C 180,E1 -30645.138,E2 -30645.138} C_VEL
LIN {X 0,Y 217.652,Z 543.038,A -85,B 0,C 180,E1 -30646.861,E2 -30646.861} C_VEL
LIN {X 0,Y 212.08,Z 553.318,A -85,B 0,C 180,E1 -30648.665,E2 -30648.665} C_VEL
LIN {X 0,Y 205.938,Z 563.579,A -85,B 0,C 180,E1 -30651.014,E2 -30651.014} C_VEL
LIN {X 0,Y 200.158,Z 572.094,A -85,B 0,C 180,E1 -30653.501,E2 -30653.501} C_VEL
LIN {X 0,Y 193.915,Z 580.28,A -85,B 0,C 180,E1 -30656.581,E2 -30656.581} C_VEL
LIN {X 0,Y 188.4,Z 586.917,A -85,B 0,C 180,E1 -30659.88,E2 -30659.88} C_VEL
LIN {X 0,Y 183.346,Z 592.505,A -85,B 0,C 180,E1 -30663.617,E2 -30663.617} C_VEL
LIN {X 0,Y 180.895,Z 594.498,A -85,B 0,C 180,E1 -30665.193,E2 -30665.193} C_VEL
LIN {X 0,Y 175.473,Z 597.161,A -85,B 0,C 180,E1 -30667.723,E2 -30667.723} C_VEL
LIN {X 0,Y 171.257,Z 598.859,A -85,B 0,C 180,E1 -30669.88,E2 -30669.88} C_VEL
LIN {X 0,Y 168.975,Z 599.898,A -85,B 0,C 180,E1 -30671.684,E2 -30671.684} C_VEL
LIN {X 0,Y 168.501,Z 600.19,A -85,B 0,C 180,E1 -30672.324,E2 -30672.324} C_VEL
LIN {X 0,Y 166.986,Z 601.357,A -85,B 0,C 180,E1 -30675.429,E2 -30675.429} C_VEL
LIN {X 0,Y 165.579,Z 602.024,A -85,B 0,C 180,E1 -30680.264,E2 -30680.264} C_VEL
LIN {X 0,Y 165.398,Z 601.412,A -85,B 0,C 180,E1 -30685.147,E2 -30685.147} C_VEL
LIN {X 0,Y 166.294,Z 599.492,A -85,B 0,C 180,E1 -30690.006,E2 -30690.006} C_VEL
LIN {X 0,Y 167.516,Z 596.766,A -85,B 0,C 180,E1 -30694.352,E2 -30694.352} C_VEL
LIN {X 0,Y 167.234,Z 602.523,A -85,B 0,C 180,E1 -30698.435,E2 -30698.435} C_VEL
LIN {X 0,Y 167.93,Z 607.977,A -85,B 0,C 180,E1 -30703.268,E2 -30703.268} C_VEL
LIN {X 0,Y 169.421,Z 611.268,A -85,B 0,C 180,E1 -30706.828,E2 -30706.828} C_VEL
LIN {X 0,Y 172.737,Z 614.603,A -85,B 0,C 180,E1 -30711.41,E2 -30711.41} C_VEL
LIN {X 0,Y 177.209,Z 616.793,A -85,B 0,C 180,E1 -30715.778,E2 -30715.778} C_VEL
LIN {X 0,Y 183.013,Z 617.922,A -85,B 0,C 180,E1 -30719.843,E2 -30719.843} C_VEL
LIN {X 0,Y 190.047,Z 617.979,A -85,B 0,C 180,E1 -30723.568,E2 -30723.568} C_VEL
LIN {X 0,Y 197.846,Z 616.957,A -85,B 0,C 180,E1 -30727.009,E2 -30727.009} C_VEL
LIN {X 0,Y 206.666,Z 614.833,A -85,B 0,C 180,E1 -30730.093,E2 -30730.093} C_VEL
LIN {X 0,Y 216.295,Z 611.544,A -85,B 0,C 180,E1 -30732.853,E2 -30732.853} C_VEL
LIN {X 0,Y 226.647,Z 606.99,A -85,B 0,C 180,E1 -30735.306,E2 -30735.306} C_VEL
LIN {X 0,Y 237.507,Z 601.1,A -85,B 0,C 180,E1 -30737.506,E2 -30737.506} C_VEL
LIN {X 0,Y 246.868,Z 595.151,A -85,B 0,C 180,E1 -30739.115,E2 -30739.115} C_VEL
LIN {X 0,Y 257.854,Z 586.971,A -85,B 0,C 180,E1 -30740.736,E2 -30740.736} C_VEL
LIN {X 0,Y 260.907,Z 584.442,A -85,B 0,C 180,E1 -30741.133,E2 -30741.133} C_VEL
LIN {X 0,Y 261.66,Z 583.784,A -85,B 0,C 180,E1 -30741.633,E2 -30741.633} C_VEL
LIN {X 0,Y 251.265,Z 591.723,A -85,B 0,C 180,E1 -30743.177,E2 -30743.177} C_VEL
LIN {X 0,Y 242.355,Z 597.59,A -85,B 0,C 180,E1 -30744.688,E2 -30744.688} C_VEL
LIN {X 0,Y 230.97,Z 603.861,A -85,B 0,C 180,E1 -30746.916,E2 -30746.916} C_VEL
LIN {X 0,Y 220.265,Z 608.576,A -85,B 0,C 180,E1 -30749.416,E2 -30749.416} C_VEL
LIN {X 0,Y 210.264,Z 611.92,A -85,B 0,C 180,E1 -30752.201,E2 -30752.201} C_VEL
LIN {X 0,Y 200.973,Z 614.004,A -85,B 0,C 180,E1 -30755.277,E2 -30755.277} C_VEL
LIN {X 0,Y 192.584,Z 614.874,A -85,B 0,C 180,E1 -30758.672,E2 -30758.672} C_VEL
LIN {X 0,Y 185.137,Z 614.563,A -85,B 0,C 180,E1 -30762.382,E2 -30762.382} C_VEL
LIN {X 0,Y 178.89,Z 613.095,A -85,B 0,C 180,E1 -30766.412,E2 -30766.412} C_VEL
LIN {X 0,Y 173.909,Z 610.485,A -85,B 0,C 180,E1 -30770.729,E2 -30770.729} C_VEL
LIN {X 0,Y 170.231,Z 606.711,A -85,B 0,C 180,E1 -30775.28,E2 -30775.28} C_VEL
LIN {X 0,Y 167.851,Z 601.569,A -85,B 0,C 180,E1 -30780.11,E2 -30780.11} C_VEL
LIN {X 0,Y 166.636,Z 595.253,A -85,B 0,C 180,E1 -30784.822,E2 -30784.822} C_VEL
LIN {X 0,Y 166.434,Z 588.273,A -85,B 0,C 180,E1 -30789.08,E2 -30789.08} C_VEL
LIN {X 0,Y 166.668,Z 579.583,A -85,B 0,C 180,E1 -30793.364,E2 -30793.364} C_VEL
LIN {X 0,Y 167.011,Z 570.305,A -85,B 0,C 180,E1 -30797.072,E2 -30797.072} C_VEL
LIN {X 0,Y 167.492,Z 559.903,A -85,B 0,C 180,E1 -30800.502,E2 -30800.502} C_VEL
LIN {X 0,Y 168.223,Z 548.45,A -85,B 0,C 180,E1 -30803.635,E2 -30803.635} C_VEL
LIN {X 0,Y 169.137,Z 535.959,A -85,B 0,C 180,E1 -30806.435,E2 -30806.435} C_VEL
LIN {X 0,Y 170.265,Z 522.33,A -85,B 0,C 180,E1 -30808.906,E2 -30808.906} C_VEL
LIN {X 0,Y 171.293,Z 508.428,A -85,B 0,C 180,E1 -30810.891,E2 -30810.891} C_VEL
LIN {X 0,Y 172.298,Z 493.23,A -85,B 0,C 180,E1 -30812.549,E2 -30812.549} C_VEL
LIN {X 0,Y 173.277,Z 476.428,A -85,B 0,C 180,E1 -30813.854,E2 -30813.854} C_VEL
LIN {X 0,Y 177.311,Z 393.596,A -85,B 0,C 180,E1 -30819.564,E2 -30819.564} C_VEL
LIN {X 0,Y 174.904,Z 365.358,A -85,B 0,C 180,E1 -30821.57,E2 -30821.57} C_VEL
LIN {X 0,Y 171.082,Z 348.384,A -85,B 0,C 180,E1 -30822.948,E2 -30822.948} C_VEL
LIN {X 0,Y 168.607,Z 336.035,A -85,B 0,C 180,E1 -30826.925,E2 -30826.925} C_VEL
LIN {X 0,Y 168.495,Z 336.227,A -85,B 0,C 180,E1 -30831.802,E2 -30831.802} C_VEL
LIN {X 0,Y 169.43,Z 338.84,A -85,B 0,C 180,E1 -30832.273,E2 -30832.273} C_VEL
LIN {X 0,Y 171.677,Z 341.527,A -85,B 0,C 180,E1 -30833.164,E2 -30833.164} C_VEL
LIN {X 0,Y 173.941,Z 344.918,A -85,B 0,C 180,E1 -30834.064,E2 -30834.064} C_VEL
LIN {X 0,Y 181.592,Z 356.928,A -85,B 0,C 180,E1 -30836.894,E2 -30836.894} C_VEL
LIN {X 0,Y 188.791,Z 369.973,A -85,B 0,C 180,E1 -30839.338,E2 -30839.338} C_VEL
LIN {X 0,Y 195.595,Z 384.351,A -85,B 0,C 180,E1 -30841.511,E2 -30841.511} C_VEL
LIN {X 0,Y 196.576,Z 387.383,A -85,B 0,C 180,E1 -30841.85,E2 -30841.85} C_VEL
LIN {X 0,Y 192.644,Z 458.539,A -85,B 0,C 180,E1 -30844.27,E2 -30844.27} C_VEL
LIN {X 0,Y 191.222,Z 472.913,A -85,B 0,C 180,E1 -30845.154,E2 -30845.154} C_VEL
LIN {X 0,Y 189.292,Z 486.715,A -85,B 0,C 180,E1 -30846.41,E2 -30846.41} C_VEL
LIN {X 0,Y 186.905,Z 499.608,A -85,B 0,C 180,E1 -30847.985,E2 -30847.985} C_VEL
LIN {X 0,Y 183.811,Z 512.209,A -85,B 0,C 180,E1 -30849.937,E2 -30849.937} C_VEL
LIN {X 0,Y 180.741,Z 523.662,A -85,B 0,C 180,E1 -30852.225,E2 -30852.225} C_VEL
LIN {X 0,Y 178.13,Z 533.165,A -85,B 0,C 180,E1 -30854.602,E2 -30854.602} C_VEL
LIN {X 0,Y 174.727,Z 543.794,A -85,B 0,C 180,E1 -30857.845,E2 -30857.845} C_VEL
LIN {X 0,Y 172.023,Z 552.542,A -85,B 0,C 180,E1 -30861.211,E2 -30861.211} C_VEL
LIN {X 0,Y 169.672,Z 559.844,A -85,B 0,C 180,E1 -30864.665,E2 -30864.665} C_VEL
LIN {X 0,Y 167.903,Z 566.802,A -85,B 0,C 180,E1 -30868.798,E2 -30868.798} C_VEL
LIN {X 0,Y 166.692,Z 571.666,A -85,B 0,C 180,E1 -30872.402,E2 -30872.402} C_VEL
LIN {X 0,Y 165.563,Z 576.732,A -85,B 0,C 180,E1 -30877.286,E2 -30877.286} C_VEL
LIN {X 0,Y 165.456,Z 580.289,A -85,B 0,C 180,E1 -30882.214,E2 -30882.214} C_VEL
LIN {X 0,Y 165.993,Z 582.467,A -85,B 0,C 180,E1 -30887.174,E2 -30887.174} C_VEL
LIN {X 0,Y 167.527,Z 583.272,A -85,B 0,C 180,E1 -30892.098,E2 -30892.098} C_VEL
LIN {X 0,Y 170.034,Z 582.696,A -85,B 0,C 180,E1 -30896.938,E2 -30896.938} C_VEL
LIN {X 0,Y 173.563,Z 580.722,A -85,B 0,C 180,E1 -30901.637,E2 -30901.637} C_VEL
LIN {X 0,Y 178.079,Z 577.297,A -85,B 0,C 180,E1 -30906.15,E2 -30906.15} C_VEL
LIN {X 0,Y 183.612,Z 572.305,A -85,B 0,C 180,E1 -30910.422,E2 -30910.422} C_VEL
LIN {X 0,Y 188.306,Z 567.415,A -85,B 0,C 180,E1 -30913.476,E2 -30913.476} C_VEL
LIN {X 0,Y 194.312,Z 560.459,A -85,B 0,C 180,E1 -30916.772,E2 -30916.772} C_VEL
LIN {X 0,Y 200.136,Z 552.803,A -85,B 0,C 180,E1 -30919.563,E2 -30919.563} C_VEL
LIN {X 0,Y 205.977,Z 544.214,A -85,B 0,C 180,E1 -30922.001,E2 -30922.001} C_VEL
LIN {X 0,Y 211.678,Z 534.635,A -85,B 0,C 180,E1 -30924.156,E2 -30924.156} C_VEL
LIN {X 0,Y 217.265,Z 523.713,A -85,B 0,C 180,E1 -30926.106,E2 -30926.106} C_VEL
LIN {X 0,Y 222.32,Z 512.098,A -85,B 0,C 180,E1 -30927.731,E2 -30927.731} C_VEL
LIN {X 0,Y 226.602,Z 500.122,A -85,B 0,C 180,E1 -30929.058,E2 -30929.058} C_VEL
LIN {X 0,Y 230.144,Z 487.618,A -85,B 0,C 180,E1 -30930.147,E2 -30930.147} C_VEL
LIN {X 0,Y 233.273,Z 473.161,A -85,B 0,C 180,E1 -30931.068,E2 -30931.068} C_VEL
LIN {X 0,Y 235.32,Z 458.976,A -85,B 0,C 180,E1 -30931.673,E2 -30931.673} C_VEL
LIN {X 0,Y 237.995,Z 425.411,A -85,B 0,C 180,E1 -30932.573,E2 -30932.573} C_VEL
LIN {X 0,Y 232.692,Z 415.125,A -85,B 0,C 180,E1 -30935.198,E2 -30935.198} C_VEL
LIN {X 0,Y 227.124,Z 405.441,A -85,B 0,C 180,E1 -30938.28,E2 -30938.28} C_VEL
LIN {X 0,Y 222.477,Z 398.041,A -85,B 0,C 180,E1 -30941.203,E2 -30941.203} C_VEL
LIN {X 0,Y 218.359,Z 391.638,A -85,B 0,C 180,E1 -30944.203,E2 -30944.203} C_VEL
LIN {X 0,Y 215.093,Z 387.145,A -85,B 0,C 180,E1 -30946.937,E2 -30946.937} C_VEL
LIN {X 0,Y 212.06,Z 382.739,A -85,B 0,C 180,E1 -30950.014,E2 -30950.014} C_VEL
LIN {X 0,Y 209.789,Z 379.809,A -85,B 0,C 180,E1 -30952.823,E2 -30952.823} C_VEL
LIN {X 0,Y 208.91,Z 377.954,A -85,B 0,C 180,E1 -30954.227,E2 -30954.227} C_VEL
LIN {X 0,Y 206.565,Z 375.374,A -85,B 0,C 180,E1 -30958.725,E2 -30958.725} C_VEL
LIN {X 0,Y 205.778,Z 372.823,A -85,B 0,C 180,E1 -30961.951,E2 -30961.951} C_VEL
LIN {X 0,Y 205.538,Z 373.042,A -85,B 0,C 180,E1 -30968.241,E2 -30968.241} C_VEL
LIN {X 0,Y 207.236,Z 377.181,A -85,B 0,C 180,E1 -30974.309,E2 -30974.309} C_VEL
LIN {X 0,Y 209.781,Z 381.211,A -85,B 0,C 180,E1 -30978.634,E2 -30978.634} C_VEL
LIN {X 0,Y 213.565,Z 387.974,A -85,B 0,C 180,E1 -30983.177,E2 -30983.177} C_VEL
LIN {X 0,Y 217.042,Z 394.185,A -85,B 0,C 180,E1 -30986.391,E2 -30986.391} C_VEL
LIN {X 0,Y 219.906,Z 399.426,A -85,B 0,C 180,E1 -30988.67,E2 -30988.67} C_VEL
LIN {X 0,Y 223.495,Z 406.438,A -85,B 0,C 180,E1 -30991.221,E2 -30991.221} C_VEL
LIN {X 0,Y 227.906,Z 415.79,A -85,B 0,C 180,E1 -30994.02,E2 -30994.02} C_VEL
LIN {X 0,Y 232.812,Z 427.465,A -85,B 0,C 180,E1 -30996.83,E2 -30996.83} C_VEL
LIN {X 0,Y 236.737,Z 438.054,A -85,B 0,C 180,E1 -30998.903,E2 -30998.903} C_VEL
LIN {X 0,Y 237.03,Z 438.948,A -85,B 0,C 180,E1 -30999.056,E2 -30999.056} C_VEL
LIN {X 0,Y 233.912,Z 476.151,A -85,B 0,C 180,E1 -31000.027,E2 -31000.027} C_VEL
LIN {X 0,Y 231.421,Z 490.955,A -85,B 0,C 180,E1 -31000.615,E2 -31000.615} C_VEL
LIN {X 0,Y 227.91,Z 505.497,A -85,B 0,C 180,E1 -31001.493,E2 -31001.493} C_VEL
LIN {X 0,Y 223.393,Z 519.008,A -85,B 0,C 180,E1 -31002.545,E2 -31002.545} C_VEL
LIN {X 0,Y 218.432,Z 531.176,A -85,B 0,C 180,E1 -31003.828,E2 -31003.828} C_VEL
LIN {X 0,Y 212.547,Z 543.483,A -85,B 0,C 180,E1 -31005.557,E2 -31005.557} C_VEL
LIN {X 0,Y 206.828,Z 553.631,A -85,B 0,C 180,E1 -31007.373,E2 -31007.373} C_VEL
LIN {X 0,Y 200.477,Z 563.736,A -85,B 0,C 180,E1 -31009.739,E2 -31009.739} C_VEL
LIN {X 0,Y 194.49,Z 572.162,A -85,B 0,C 180,E1 -31012.255,E2 -31012.255} C_VEL
LIN {X 0,Y 188.027,Z 580.247,A -85,B 0,C 180,E1 -31015.389,E2 -31015.389} C_VEL
LIN {X 0,Y 182.263,Z 586.805,A -85,B 0,C 180,E1 -31018.754,E2 -31018.754} C_VEL
LIN {X 0,Y 176.663,Z 592.678,A -85,B 0,C 180,E1 -31022.88,E2 -31022.88} C_VEL
LIN {X 0,Y 173.219,Z 596.114,A -85,B 0,C 180,E1 -31026.155,E2 -31026.155} C_VEL
LIN {X 0,Y 169.533,Z 599.4,A -85,B 0,C 180,E1 -31030.706,E2 -31030.706} C_VEL
LIN {X 0,Y 168.501,Z 600.19,A -85,B 0,C 180,E1 -31032.324,E2 -31032.324} C_VEL
LIN {X 0,Y 166.791,Z 600.983,A -85,B 0,C 180,E1 -31034.24,E2 -31034.24} C_VEL
LIN {X 0,Y 162.641,Z 601.667,A -85,B 0,C 180,E1 -31037.369,E2 -31037.369} C_VEL
LIN {X 0,Y 159.032,Z 601.647,A -85,B 0,C 180,E1 -31040.663,E2 -31040.663} C_VEL
LIN {X 0,Y 158.213,Z 601.337,A -85,B 0,C 180,E1 -31042.775,E2 -31042.775} C_VEL
LIN {X 0,Y 158.669,Z 600.102,A -85,B 0,C 180,E1 -31047.476,E2 -31047.476} C_VEL
LIN {X 0,Y 159.904,Z 597.435,A -85,B 0,C 180,E1 -31052.517,E2 -31052.517} C_VEL
LIN {X 0,Y 160.681,Z 595.515,A -85,B 0,C 180,E1 -31055.164,E2 -31055.164} C_VEL
LIN {X 0,Y 160.5,Z 602.137,A -85,B 0,C 180,E1 -31060.059,E2 -31060.059} C_VEL
LIN {X 0,Y 161.614,Z 607.571,A -85,B 0,C 180,E1 -31065.079,E2 -31065.079} C_VEL
LIN {X 0,Y 164.362,Z 611.811,A -85,B 0,C 180,E1 -31069.939,E2 -31069.939} C_VEL
LIN {X 0,Y 168.41,Z 614.886,A -85,B 0,C 180,E1 -31074.583,E2 -31074.583} C_VEL
LIN {X 0,Y 173.717,Z 616.879,A -85,B 0,C 180,E1 -31078.943,E2 -31078.943} C_VEL
LIN {X 0,Y 180.383,Z 617.817,A -85,B 0,C 180,E1 -31082.937,E2 -31082.937} C_VEL
LIN {X 0,Y 188.17,Z 617.668,A -85,B 0,C 180,E1 -31086.56,E2 -31086.56} C_VEL
LIN {X 0,Y 192.228,Z 617.196,A -85,B 0,C 180,E1 -31088.282,E2 -31088.282} C_VEL
LIN {X 0,Y 201.32,Z 615.44,A -85,B 0,C 180,E1 -31091.386,E2 -31091.386} C_VEL
LIN {X 0,Y 211.204,Z 612.555,A -85,B 0,C 180,E1 -31094.148,E2 -31094.148} C_VEL
LIN {X 0,Y 221.78,Z 608.469,A -85,B 0,C 180,E1 -31096.591,E2 -31096.591} C_VEL
LIN {X 0,Y 232.892,Z 603.094,A -85,B 0,C 180,E1 -31098.76,E2 -31098.76} C_VEL
LIN {X 0,Y 244.533,Z 596.27,A -85,B 0,C 180,E1 -31100.665,E2 -31100.665} C_VEL
LIN {X 0,Y 247.131,Z 594.59,A -85,B 0,C 180,E1 -31101.046,E2 -31101.046} C_VEL
LIN {X 0,Y 248.717,Z 593.454,A -85,B 0,C 180,E1 -31101.715,E2 -31101.715} C_VEL
LIN {X 0,Y 239.535,Z 599.067,A -85,B 0,C 180,E1 -31103.169,E2 -31103.169} C_VEL
LIN {X 0,Y 227.828,Z 605.031,A -85,B 0,C 180,E1 -31105.335,E2 -31105.335} C_VEL
LIN {X 0,Y 219.474,Z 608.531,A -85,B 0,C 180,E1 -31107.143,E2 -31107.143} C_VEL
LIN {X 0,Y 208.923,Z 611.956,A -85,B 0,C 180,E1 -31109.808,E2 -31109.808} C_VEL
LIN {X 0,Y 199.051,Z 614.124,A -85,B 0,C 180,E1 -31112.777,E2 -31112.777} C_VEL
LIN {X 0,Y 190.037,Z 615.084,A -85,B 0,C 180,E1 -31116.081,E2 -31116.081} C_VEL
LIN {X 0,Y 181.916,Z 614.866,A -85,B 0,C 180,E1 -31119.724,E2 -31119.724} C_VEL
LIN {X 0,Y 174.928,Z 613.486,A -85,B 0,C 180,E1 -31123.722,E2 -31123.722} C_VEL
LIN {X 0,Y 169.247,Z 610.982,A -85,B 0,C 180,E1 -31128.057,E2 -31128.057} C_VEL
LIN {X 0,Y 164.835,Z 607.335,A -85,B 0,C 180,E1 -31132.676,E2 -31132.676} C_VEL
LIN {X 0,Y 161.571,Z 601.677,A -85,B 0,C 180,E1 -31138.285,E2 -31138.285} C_VEL
LIN {X 0,Y 159.945,Z 594.567,A -85,B 0,C 180,E1 -31143.766,E2 -31143.766} C_VEL
LIN {X 0,Y 159.639,Z 586.357,A -85,B 0,C 180,E1 -31148.834,E2 -31148.834} C_VEL
LIN {X 0,Y 159.834,Z 578.745,A -85,B 0,C 180,E1 -31152.657,E2 -31152.657} C_VEL
LIN {X 0,Y 160.121,Z 569.389,A -85,B 0,C 180,E1 -31156.518,E2 -31156.518} C_VEL
LIN {X 0,Y 160.574,Z 558.896,A -85,B 0,C 180,E1 -31160.091,E2 -31160.091} C_VEL
LIN {X 0,Y 161.291,Z 546.945,A -85,B 0,C 180,E1 -31163.44,E2 -31163.44} C_VEL
LIN {X 0,Y 162.194,Z 534.602,A -85,B 0,C 180,E1 -31166.273,E2 -31166.273} C_VEL
LIN {X 0,Y 163.304,Z 520.674,A -85,B 0,C 180,E1 -31168.851,E2 -31168.851} C_VEL
LIN {X 0,Y 164.252,Z 507.462,A -85,B 0,C 180,E1 -31170.779,E2 -31170.779} C_VEL
LIN {X 0,Y 165.238,Z 492.332,A -85,B 0,C 180,E1 -31172.469,E2 -31172.469} C_VEL
LIN {X 0,Y 166.417,Z 472.02,A -85,B 0,C 180,E1 -31174.078,E2 -31174.078} C_VEL
LIN {X 0,Y 170.232,Z 393.434,A -85,B 0,C 180,E1 -31179.769,E2 -31179.769} C_VEL
LIN {X 0,Y 167.897,Z 366.428,A -85,B 0,C 180,E1 -31181.772,E2 -31181.772} C_VEL
LIN {X 0,Y 163.89,Z 348.545,A -85,B 0,C 180,E1 -31183.271,E2 -31183.271} C_VEL
LIN {X 0,Y 161.583,Z 336.911,A -85,B 0,C 180,E1 -31187.108,E2 -31187.108} C_VEL
LIN {X 0,Y 161.422,Z 336.928,A -85,B 0,C 180,E1 -31189.253,E2 -31189.253} C_VEL
LIN {X 0,Y 162.331,Z 339.657,A -85,B 0,C 180,E1 -31189.792,E2 -31189.792} C_VEL
LIN {X 0,Y 164.76,Z 342.493,A -85,B 0,C 180,E1 -31190.872,E2 -31190.872} C_VEL
LIN {X 0,Y 166.908,Z 345.73,A -85,B 0,C 180,E1 -31191.827,E2 -31191.827} C_VEL
LIN {X 0,Y 171.329,Z 352.285,A -85,B 0,C 180,E1 -31193.668,E2 -31193.668} C_VEL
LIN {X 0,Y 177.403,Z 362.003,A -85,B 0,C 180,E1 -31196.011,E2 -31196.011} C_VEL
LIN {X 0,Y 184.018,Z 374.204,A -85,B 0,C 180,E1 -31198.388,E2 -31198.388} C_VEL
LIN {X 0,Y 190.598,Z 388.41,A -85,B 0,C 180,E1 -31200.616,E2 -31200.616} C_VEL
LIN {X 0,Y 189.993,Z 402.604,A -85,B 0,C 180,E1 -31201.139,E2 -31201.139} C_VEL
LIN {X 0,Y 186.715,Z 458.857,A -85,B 0,C 180,E1 -31203.099,E2 -31203.099} C_VEL
LIN {X 0,Y 185.239,Z 473.171,A -85,B 0,C 180,E1 -31203.993,E2 -31203.993} C_VEL
LIN {X 0,Y 183.245,Z 487.007,A -85,B 0,C 180,E1 -31205.281,E2 -31205.281} C_VEL
LIN {X 0,Y 180.761,Z 499.927,A -85,B 0,C 180,E1 -31206.894,E2 -31206.894} C_VEL
LIN {X 0,Y 177.538,Z 512.549,A -85,B 0,C 180,E1 -31208.894,E2 -31208.894} C_VEL
LIN {X 0,Y 174.36,Z 524.011,A -85,B 0,C 180,E1 -31211.248,E2 -31211.248} C_VEL
LIN {X 0,Y 171.933,Z 532.554,A -85,B 0,C 180,E1 -31213.425,E2 -31213.425} C_VEL
LIN {X 0,Y 168.323,Z 543.355,A -85,B 0,C 180,E1 -31216.764,E2 -31216.764} C_VEL
LIN {X 0,Y 165.46,Z 552.244,A -85,B 0,C 180,E1 -31220.245,E2 -31220.245} C_VEL
LIN {X 0,Y 162.922,Z 559.675,A -85,B 0,C 180,E1 -31223.824,E2 -31223.824} C_VEL
LIN {X 0,Y 161.247,Z 565.927,A -85,B 0,C 180,E1 -31227.567,E2 -31227.567} C_VEL
LIN {X 0,Y 159.931,Z 570.964,A -85,B 0,C 180,E1 -31231.249,E2 -31231.249} C_VEL
LIN {X 0,Y 158.872,Z 575.11,A -85,B 0,C 180,E1 -31235.052,E2 -31235.052} C_VEL
LIN {X 0,Y 158.313,Z 579.323,A -85,B 0,C 180,E1 -31240.187,E2 -31240.187} C_VEL
LIN {X 0,Y 158.458,Z 581.245,A -85,B 0,C 180,E1 -31243.472,E2 -31243.472} C_VEL
LIN {X 0,Y 159.047,Z 582.981,A -85,B 0,C 180,E1 -31247.949,E2 -31247.949} C_VEL
LIN {X 0,Y 160.797,Z 583.687,A -85,B 0,C 180,E1 -31253.075,E2 -31253.075} C_VEL
LIN {X 0,Y 163.525,Z 583.026,A -85,B 0,C 180,E1 -31258.103,E2 -31258.103} C_VEL
LIN {X 0,Y 167.372,Z 580.973,A -85,B 0,C 180,E1 -31262.952,E2 -31262.952} C_VEL
LIN {X 0,Y 172.216,Z 577.466,A -85,B 0,C 180,E1 -31267.588,E2 -31267.588} C_VEL
LIN {X 0,Y 178.088,Z 572.387,A -85,B 0,C 180,E1 -31271.953,E2 -31271.953} C_VEL
LIN {X 0,Y 183.057,Z 567.404,A -85,B 0,C 180,E1 -31275.054,E2 -31275.054} C_VEL
LIN {X 0,Y 188.838,Z 560.991,A -85,B 0,C 180,E1 -31278.113,E2 -31278.113} C_VEL
LIN {X 0,Y 195.458,Z 552.575,A -85,B 0,C 180,E1 -31281.2,E2 -31281.2} C_VEL
LIN {X 0,Y 201.689,Z 543.641,A -85,B 0,C 180,E1 -31283.696,E2 -31283.696} C_VEL
LIN {X 0,Y 208.055,Z 533.126,A -85,B 0,C 180,E1 -31285.99,E2 -31285.99} C_VEL
LIN {X 0,Y 213.875,Z 521.8,A -85,B 0,C 180,E1 -31287.921,E2 -31287.921} C_VEL
LIN {X 0,Y 219.285,Z 509.161,A -85,B 0,C 180,E1 -31289.581,E2 -31289.581} C_VEL
LIN {X 0,Y 223.523,Z 496.84,A -85,B 0,C 180,E1 -31290.858,E2 -31290.858} C_VEL
LIN {X 0,Y 226.908,Z 484.514,A -85,B 0,C 180,E1 -31291.837,E2 -31291.837} C_VEL
LIN {X 0,Y 229.74,Z 470.465,A -85,B 0,C 180,E1 -31292.663,E2 -31292.663} C_VEL
LIN {X 0,Y 231.641,Z 456.491,A -85,B 0,C 180,E1 -31293.186,E2 -31293.186} C_VEL
LIN {X 0,Y 233.915,Z 428.694,A -85,B 0,C 180,E1 -31293.917,E2 -31293.917} C_VEL
LIN {X 0,Y 228.829,Z 418.649,A -85,B 0,C 180,E1 -31296.634,E2 -31296.634} C_VEL
LIN {X 0,Y 223.79,Z 409.761,A -85,B 0,C 180,E1 -31299.638,E2 -31299.638} C_VEL
LIN {X 0,Y 218.995,Z 401.938,A -85,B 0,C 180,E1 -31302.926,E2 -31302.926} C_VEL
LIN {X 0,Y 215.813,Z 397.196,A -85,B 0,C 180,E1 -31305.432,E2 -31305.432} C_VEL
LIN {X 0,Y 213.478,Z 393.687,A -85,B 0,C 180,E1 -31307.532,E2 -31307.532} C_VEL
LIN {X 0,Y 210.752,Z 389.548,A -85,B 0,C 180,E1 -31310.434,E2 -31310.434} C_VEL
LIN {X 0,Y 208.443,Z 386.411,A -85,B 0,C 180,E1 -31313.443,E2 -31313.443} C_VEL
LIN {X 0,Y 207.796,Z 384.882,A -85,B 0,C 180,E1 -31314.553,E2 -31314.553} C_VEL
LIN {X 0,Y 205.5,Z 382.199,A -85,B 0,C 180,E1 -31319.222,E2 -31319.222} C_VEL
LIN {X 0,Y 204.892,Z 379.939,A -85,B 0,C 180,E1 -31321.959,E2 -31321.959} C_VEL
LIN {X 0,Y 204.646,Z 380.079,A -85,B 0,C 180,E1 -31328.13,E2 -31328.13} C_VEL
LIN {X 0,Y 206.194,Z 384.171,A -85,B 0,C 180,E1 -31334.007,E2 -31334.007} C_VEL
LIN {X 0,Y 208.484,Z 387.95,A -85,B 0,C 180,E1 -31338.106,E2 -31338.106} C_VEL
LIN {X 0,Y 212.045,Z 394.626,A -85,B 0,C 180,E1 -31342.624,E2 -31342.624} C_VEL
LIN {X 0,Y 215.124,Z 400.351,A -85,B 0,C 180,E1 -31345.623,E2 -31345.623} C_VEL
LIN {X 0,Y 218.069,Z 406.071,A -85,B 0,C 180,E1 -31348.095,E2 -31348.095} C_VEL
LIN {X 0,Y 221.519,Z 413.115,A -85,B 0,C 180,E1 -31350.656,E2 -31350.656} C_VEL
LIN {X 0,Y 225.749,Z 422.641,A -85,B 0,C 180,E1 -31353.467,E2 -31353.467} C_VEL
LIN {X 0,Y 230.178,Z 433.737,A -85,B 0,C 180,E1 -31356.128,E2 -31356.128} C_VEL
LIN {X 0,Y 232.937,Z 441.569,A -85,B 0,C 180,E1 -31357.684,E2 -31357.684} C_VEL
LIN {X 0,Y 229.929,Z 475.841,A -85,B 0,C 180,E1 -31358.571,E2 -31358.571} C_VEL
LIN {X 0,Y 227.412,Z 490.486,A -85,B 0,C 180,E1 -31359.15,E2 -31359.15} C_VEL
LIN {X 0,Y 223.924,Z 504.561,A -85,B 0,C 180,E1 -31359.979,E2 -31359.979} C_VEL
LIN {X 0,Y 219.329,Z 518.177,A -85,B 0,C 180,E1 -31361.028,E2 -31361.028} C_VEL
LIN {X 0,Y 214.226,Z 530.425,A -85,B 0,C 180,E1 -31362.297,E2 -31362.297} C_VEL
LIN {X 0,Y 208.11,Z 542.813,A -85,B 0,C 180,E1 -31364.001,E2 -31364.001} C_VEL
LIN {X 0,Y 201.665,Z 553.9,A -85,B 0,C 180,E1 -31366.007,E2 -31366.007} C_VEL
LIN {X 0,Y 195.117,Z 563.886,A -85,B 0,C 180,E1 -31368.392,E2 -31368.392} C_VEL
LIN {X 0,Y 188.926,Z 572.215,A -85,B 0,C 180,E1 -31370.937,E2 -31370.937} C_VEL
LIN {X 0,Y 182.23,Z 580.214,A -85,B 0,C 180,E1 -31374.122,E2 -31374.122} C_VEL
LIN {X 0,Y 176.205,Z 586.695,A -85,B 0,C 180,E1 -31377.551,E2 -31377.551} C_VEL
LIN {X 0,Y 170.342,Z 592.498,A -85,B 0,C 180,E1 -31381.786,E2 -31381.786} C_VEL
LIN {X 0,Y 166.726,Z 595.869,A -85,B 0,C 180,E1 -31385.165,E2 -31385.165} C_VEL
LIN {X 0,Y 162.821,Z 599.089,A -85,B 0,C 180,E1 -31389.877,E2 -31389.877} C_VEL
LIN {X 0,Y 160.084,Z 600.984,A -85,B 0,C 180,E1 -31394.786,E2 -31394.786} C_VEL
LIN {X 0,Y 158.575,Z 601.594,A -85,B 0,C 180,E1 -31399.83,E2 -31399.83} C_VEL
LIN {X 0,Y 158.213,Z 601.337,A -85,B 0,C 180,E1 -31402.775,E2 -31402.775} C_VEL
LIN {X 0,Y 157.624,Z 600.889,A -85,B 0,C 180,E1 -31404.898,E2 -31404.898} C_VEL
LIN {X 0,Y 155.269,Z 599.455,A -85,B 0,C 180,E1 -31408.388,E2 -31408.388} C_VEL
LIN {X 0,Y 153.51,Z 597.842,A -85,B 0,C 180,E1 -31411.223,E2 -31411.223} C_VEL
LIN {X 0,Y 153.082,Z 596.37,A -85,B 0,C 180,E1 -31413.381,E2 -31413.381} C_VEL
LIN {X 0,Y 153.216,Z 595.784,A -85,B 0,C 180,E1 -31414.099,E2 -31414.099} C_VEL
LIN {X 0,Y 153.932,Z 594.329,A -85,B 0,C 180,E1 -31416.128,E2 -31416.128} C_VEL
LIN {X 0,Y 153.815,Z 600.155,A -85,B 0,C 180,E1 -31420.501,E2 -31420.501} C_VEL
LIN {X 0,Y 154.975,Z 605.905,A -85,B 0,C 180,E1 -31425.741,E2 -31425.741} C_VEL
LIN {X 0,Y 157.819,Z 610.446,A -85,B 0,C 180,E1 -31430.804,E2 -31430.804} C_VEL
LIN {X 0,Y 162.044,Z 613.816,A -85,B 0,C 180,E1 -31435.617,E2 -31435.617} C_VEL
LIN {X 0,Y 167.583,Z 616.105,A -85,B 0,C 180,E1 -31440.11,E2 -31440.11} C_VEL
LIN {X 0,Y 174.484,Z 617.379,A -85,B 0,C 180,E1 -31444.201,E2 -31444.201} C_VEL
LIN {X 0,Y 182.529,Z 617.615,A -85,B 0,C 180,E1 -31447.885,E2 -31447.885} C_VEL
LIN {X 0,Y 186.708,Z 617.339,A -85,B 0,C 180,E1 -31449.631,E2 -31449.631} C_VEL
LIN {X 0,Y 196.069,Z 615.971,A -85,B 0,C 180,E1 -31452.753,E2 -31452.753} C_VEL
LIN {X 0,Y 206.201,Z 613.494,A -85,B 0,C 180,E1 -31455.514,E2 -31455.514} C_VEL
LIN {X 0,Y 217.028,Z 609.852,A -85,B 0,C 180,E1 -31457.934,E2 -31457.934} C_VEL
LIN {X 0,Y 228.366,Z 604.974,A -85,B 0,C 180,E1 -31460.073,E2 -31460.073} C_VEL
LIN {X 0,Y 234.209,Z 602.037,A -85,B 0,C 180,E1 -31461.045,E2 -31461.045} C_VEL
LIN {X 0,Y 236.908,Z 600.563,A -85,B 0,C 180,E1 -31461.619,E2 -31461.619} C_VEL
LIN {X 0,Y 224.863,Z 606.24,A -85,B 0,C 180,E1 -31463.712,E2 -31463.712} C_VEL
LIN {X 0,Y 213.449,Z 610.427,A -85,B 0,C 180,E1 -31466.092,E2 -31466.092} C_VEL
LIN {X 0,Y 202.69,Z 613.283,A -85,B 0,C 180,E1 -31468.777,E2 -31468.777} C_VEL
LIN {X 0,Y 192.628,Z 614.909,A -85,B 0,C 180,E1 -31471.789,E2 -31471.789} C_VEL
LIN {X 0,Y 183.419,Z 615.346,A -85,B 0,C 180,E1 -31475.161,E2 -31475.161} C_VEL
LIN {X 0,Y 175.157,Z 614.626,A -85,B 0,C 180,E1 -31478.906,E2 -31478.906} C_VEL
LIN {X 0,Y 168.068,Z 612.782,A -85,B 0,C 180,E1 -31483.038,E2 -31483.038} C_VEL
LIN {X 0,Y 162.283,Z 609.832,A -85,B 0,C 180,E1 -31487.537,E2 -31487.537} C_VEL
LIN {X 0,Y 157.857,Z 605.737,A -85,B 0,C 180,E1 -31492.35,E2 -31492.35} C_VEL
LIN {X 0,Y 154.956,Z 600.461,A -85,B 0,C 180,E1 -31497.409,E2 -31497.409} C_VEL
LIN {X 0,Y 153.331,Z 593.81,A -85,B 0,C 180,E1 -31502.618,E2 -31502.618} C_VEL
LIN {X 0,Y 152.836,Z 585.52,A -85,B 0,C 180,E1 -31507.902,E2 -31507.902} C_VEL
LIN {X 0,Y 153.001,Z 577.828,A -85,B 0,C 180,E1 -31511.889,E2 -31511.889} C_VEL
LIN {X 0,Y 153.285,Z 568.421,A -85,B 0,C 180,E1 -31515.913,E2 -31515.913} C_VEL
LIN {X 0,Y 153.68,Z 557.78,A -85,B 0,C 180,E1 -31519.642,E2 -31519.642} C_VEL
LIN {X 0,Y 154.336,Z 546.012,A -85,B 0,C 180,E1 -31523.044,E2 -31523.044} C_VEL
LIN {X 0,Y 155.192,Z 533.901,A -85,B 0,C 180,E1 -31525.919,E2 -31525.919} C_VEL
LIN {X 0,Y 156.289,Z 519.785,A -85,B 0,C 180,E1 -31528.619,E2 -31528.619} C_VEL
LIN {X 0,Y 157.22,Z 506.426,A -85,B 0,C 180,E1 -31530.635,E2 -31530.635} C_VEL
LIN {X 0,Y 158.188,Z 491.765,A -85,B 0,C 180,E1 -31532.323,E2 -31532.323} C_VEL
LIN {X 0,Y 159.383,Z 470.794,A -85,B 0,C 180,E1 -31534.069,E2 -31534.069} C_VEL
LIN {X 0,Y 163.111,Z 393.369,A -85,B 0,C 180,E1 -31539.95,E2 -31539.95} C_VEL
LIN {X 0,Y 160.951,Z 367.884,A -85,B 0,C 180,E1 -31541.927,E2 -31541.927} C_VEL
LIN {X 0,Y 156.649,Z 348.515,A -85,B 0,C 180,E1 -31543.647,E2 -31543.647} C_VEL
LIN {X 0,Y 154.831,Z 339.489,A -85,B 0,C 180,E1 -31546.701,E2 -31546.701} C_VEL
LIN {X 0,Y 155.704,Z 341.419,A -85,B 0,C 180,E1 -31547.221,E2 -31547.221} C_VEL
LIN {X 0,Y 157.814,Z 343.208,A -85,B 0,C 180,E1 -31548.236,E2 -31548.236} C_VEL
LIN {X 0,Y 159.812,Z 346.49,A -85,B 0,C 180,E1 -31549.262,E2 -31549.262} C_VEL
LIN {X 0,Y 161.275,Z 348.332,A -85,B 0,C 180,E1 -31549.949,E2 -31549.949} C_VEL
LIN {X 0,Y 167.026,Z 356.852,A -85,B 0,C 180,E1 -31552.534,E2 -31552.534} C_VEL
LIN {X 0,Y 173.297,Z 367.129,A -85,B 0,C 180,E1 -31555.101,E2 -31555.101} C_VEL
LIN {X 0,Y 179.451,Z 378.777,A -85,B 0,C 180,E1 -31557.445,E2 -31557.445} C_VEL
LIN {X 0,Y 184.881,Z 390.642,A -85,B 0,C 180,E1 -31559.403,E2 -31559.403} C_VEL
LIN {X 0,Y 180.852,Z 459.246,A -85,B 0,C 180,E1 -31561.856,E2 -31561.856} C_VEL
LIN {X 0,Y 179.337,Z 473.401,A -85,B 0,C 180,E1 -31562.755,E2 -31562.755} C_VEL
LIN {X 0,Y 177.278,Z 487.275,A -85,B 0,C 180,E1 -31564.076,E2 -31564.076} C_VEL
LIN {X 0,Y 174.688,Z 500.225,A -85,B 0,C 180,E1 -31565.727,E2 -31565.727} C_VEL
LIN {X 0,Y 171.329,Z 512.872,A -85,B 0,C 180,E1 -31567.774,E2 -31567.774} C_VEL
LIN {X 0,Y 168.016,Z 524.349,A -85,B 0,C 180,E1 -31570.195,E2 -31570.195} C_VEL
LIN {X 0,Y 165.131,Z 533.881,A -85,B 0,C 180,E1 -31572.721,E2 -31572.721} C_VEL
LIN {X 0,Y 161.425,Z 544.528,A -85,B 0,C 180,E1 -31576.187,E2 -31576.187} C_VEL
LIN {X 0,Y 158.43,Z 553.295,A -85,B 0,C 180,E1 -31579.808,E2 -31579.808} C_VEL
LIN {X 0,Y 155.886,Z 560.607,A -85,B 0,C 180,E1 -31583.544,E2 -31583.544} C_VEL
LIN {X 0,Y 154.172,Z 566.672,A -85,B 0,C 180,E1 -31587.39,E2 -31587.39} C_VEL
LIN {X 0,Y 152.777,Z 571.734,A -85,B 0,C 180,E1 -31591.307,E2 -31591.307} C_VEL
LIN {X 0,Y 151.473,Z 576.989,A -85,B 0,C 180,E1 -31596.632,E2 -31596.632} C_VEL
LIN {X 0,Y 151.214,Z 579.955,A -85,B 0,C 180,E1 -31600.671,E2 -31600.671} C_VEL
LIN {X 0,Y 151.385,Z 581.61,A -85,B 0,C 180,E1 -31603.676,E2 -31603.676} C_VEL
LIN {X 0,Y 152.158,Z 583.468,A -85,B 0,C 180,E1 -31608.791,E2 -31608.791} C_VEL
LIN {X 0,Y 154.129,Z 584.091,A -85,B 0,C 180,E1 -31614.135,E2 -31614.135} C_VEL
LIN {X 0,Y 157.117,Z 583.354,A -85,B 0,C 180,E1 -31619.359,E2 -31619.359} C_VEL
LIN {X 0,Y 161.334,Z 581.191,A -85,B 0,C 180,E1 -31624.422,E2 -31624.422} C_VEL
LIN {X 0,Y 166.462,Z 577.635,A -85,B 0,C 180,E1 -31629.129,E2 -31629.129} C_VEL
LIN {X 0,Y 172.717,Z 572.47,A -85,B 0,C 180,E1 -31633.576,E2 -31633.576} C_VEL
LIN {X 0,Y 177.953,Z 567.394,A -85,B 0,C 180,E1 -31636.725,E2 -31636.725} C_VEL
LIN {X 0,Y 184.715,Z 560.081,A -85,B 0,C 180,E1 -31640.155,E2 -31640.155} C_VEL
LIN {X 0,Y 190.963,Z 552.348,A -85,B 0,C 180,E1 -31642.909,E2 -31642.909} C_VEL
LIN {X 0,Y 197.521,Z 543.178,A -85,B 0,C 180,E1 -31645.432,E2 -31645.432} C_VEL
LIN {X 0,Y 204.054,Z 532.586,A -85,B 0,C 180,E1 -31647.692,E2 -31647.692} C_VEL
LIN {X 0,Y 210.078,Z 520.995,A -85,B 0,C 180,E1 -31649.613,E2 -31649.613} C_VEL
LIN {X 0,Y 215.673,Z 508.074,A -85,B 0,C 180,E1 -31651.258,E2 -31651.258} C_VEL
LIN {X 0,Y 220.046,Z 495.372,A -85,B 0,C 180,E1 -31652.525,E2 -31652.525} C_VEL
LIN {X 0,Y 223.539,Z 482.473,A -85,B 0,C 180,E1 -31653.495,E2 -31653.495} C_VEL
LIN {X 0,Y 226.341,Z 468.179,A -85,B 0,C 180,E1 -31654.277,E2 -31654.277} C_VEL
LIN {X 0,Y 228.134,Z 453.962,A -85,B 0,C 180,E1 -31654.758,E2 -31654.758} C_VEL
LIN {X 0,Y 229.903,Z 431.877,A -85,B 0,C 180,E1 -31655.353,E2 -31655.353} C_VEL
LIN {X 0,Y 225.669,Z 423.411,A -85,B 0,C 180,E1 -31657.773,E2 -31657.773} C_VEL
LIN {X 0,Y 220.846,Z 414.648,A -85,B 0,C 180,E1 -31660.849,E2 -31660.849} C_VEL
LIN {X 0,Y 216.561,Z 407.542,A -85,B 0,C 180,E1 -31663.99,E2 -31663.99} C_VEL
LIN {X 0,Y 213.747,Z 403.151,A -85,B 0,C 180,E1 -31666.362,E2 -31666.362} C_VEL
LIN {X 0,Y 211.78,Z 400.131,A -85,B 0,C 180,E1 -31668.237,E2 -31668.237} C_VEL
LIN {X 0,Y 209.278,Z 396.207,A -85,B 0,C 180,E1 -31671.065,E2 -31671.065} C_VEL
LIN {X 0,Y 206.961,Z 392.638,A -85,B 0,C 180,E1 -31674.352,E2 -31674.352} C_VEL
LIN {X 0,Y 206.467,Z 391.661,A -85,B 0,C 180,E1 -31675.235,E2 -31675.235} C_VEL
LIN {X 0,Y 204.375,Z 388.811,A -85,B 0,C 180,E1 -31680,E2 -31680} C_VEL
LIN {X 0,Y 203.91,Z 386.952,A -85,B 0,C 180,E1 -31682.461,E2 -31682.461} C_VEL
LIN {X 0,Y 203.77,Z 387.168,A -85,B 0,C 180,E1 -31688.152,E2 -31688.152} C_VEL
LIN {X 0,Y 205.168,Z 391.129,A -85,B 0,C 180,E1 -31693.714,E2 -31693.714} C_VEL
LIN {X 0,Y 207.224,Z 394.687,A -85,B 0,C 180,E1 -31697.596,E2 -31697.596} C_VEL
LIN {X 0,Y 210.365,Z 400.94,A -85,B 0,C 180,E1 -31701.858,E2 -31701.858} C_VEL
LIN {X 0,Y 213.374,Z 406.852,A -85,B 0,C 180,E1 -31704.97,E2 -31704.97} C_VEL
LIN {X 0,Y 215.899,Z 411.934,A -85,B 0,C 180,E1 -31707.21,E2 -31707.21} C_VEL
LIN {X 0,Y 219.11,Z 418.788,A -85,B 0,C 180,E1 -31709.744,E2 -31709.744} C_VEL
LIN {X 0,Y 223.01,Z 427.979,A -85,B 0,C 180,E1 -31712.501,E2 -31712.501} C_VEL
LIN {X 0,Y 227.29,Z 439.218,A -85,B 0,C 180,E1 -31715.234,E2 -31715.234} C_VEL
LIN {X 0,Y 228.965,Z 444.232,A -85,B 0,C 180,E1 -31716.255,E2 -31716.255} C_VEL
LIN {X 0,Y 226.131,Z 475.435,A -85,B 0,C 180,E1 -31717.065,E2 -31717.065} C_VEL
LIN {X 0,Y 223.642,Z 489.695,A -85,B 0,C 180,E1 -31717.621,E2 -31717.621} C_VEL
LIN {X 0,Y 220.129,Z 503.619,A -85,B 0,C 180,E1 -31718.421,E2 -31718.421} C_VEL
LIN {X 0,Y 215.427,Z 517.345,A -85,B 0,C 180,E1 -31719.455,E2 -31719.455} C_VEL
LIN {X 0,Y 210.165,Z 529.676,A -85,B 0,C 180,E1 -31720.701,E2 -31720.701} C_VEL
LIN {X 0,Y 203.89,Z 542.131,A -85,B 0,C 180,E1 -31722.395,E2 -31722.395} C_VEL
LIN {X 0,Y 197.822,Z 552.352,A -85,B 0,C 180,E1 -31724.2,E2 -31724.2} C_VEL
LIN {X 0,Y 190.971,Z 562.551,A -85,B 0,C 180,E1 -31726.559,E2 -31726.559} C_VEL
LIN {X 0,Y 184.542,Z 571.03,A -85,B 0,C 180,E1 -31729.108,E2 -31729.108} C_VEL
LIN {X 0,Y 177.786,Z 578.814,A -85,B 0,C 180,E1 -31732.119,E2 -31732.119} C_VEL
LIN {X 0,Y 171.954,Z 584.924,A -85,B 0,C 180,E1 -31735.238,E2 -31735.238} C_VEL
LIN {X 0,Y 165.521,Z 591.055,A -85,B 0,C 180,E1 -31739.489,E2 -31739.489} C_VEL
LIN {X 0,Y 160.274,Z 595.622,A -85,B 0,C 180,E1 -31744.093,E2 -31744.093} C_VEL
LIN {X 0,Y 156.147,Z 598.78,A -85,B 0,C 180,E1 -31748.977,E2 -31748.977} C_VEL
LIN {X 0,Y 153.208,Z 600.613,A -85,B 0,C 180,E1 -31754.086,E2 -31754.086} C_VEL
LIN {X 0,Y 151.566,Z 601.163,A -85,B 0,C 180,E1 -31759.354,E2 -31759.354} C_VEL
LIN {X 0,Y 151.192,Z 600.429,A -85,B 0,C 180,E1 -31764.69,E2 -31764.69} C_VEL
LIN {X 0,Y 152.125,Z 598.396,A -85,B 0,C 180,E1 -31770.006,E2 -31770.006} C_VEL
LIN {X 0,Y 153.216,Z 595.784,A -85,B 0,C 180,E1 -31774.099,E2 -31774.099} C_VEL
LIN {X 0,Y 153.229,Z 595.345,A -85,B 0,C 180,E1 -31775.522,E2 -31775.522} C_VEL
LIN {X 0,Y 152.437,Z 595.984,A -85,B 0,C 180,E1 -31777.31,E2 -31777.31} C_VEL
LIN {X 0,Y 149.458,Z 599.215,A -85,B 0,C 180,E1 -31781.192,E2 -31781.192} C_VEL
LIN {X 0,Y 147.988,Z 601.772,A -85,B 0,C 180,E1 -31784.118,E2 -31784.118} C_VEL
LIN {X 0,Y 148.083,Z 603.176,A -85,B 0,C 180,E1 -31785.585,E2 -31785.585} C_VEL
LIN {X 0,Y 150.465,Z 607.825,A -85,B 0,C 180,E1 -31790.441,E2 -31790.441} C_VEL
LIN {X 0,Y 153.408,Z 610.944,A -85,B 0,C 180,E1 -31794.27,E2 -31794.27} C_VEL
LIN {X 0,Y 158.469,Z 614.088,A -85,B 0,C 180,E1 -31799.098,E2 -31799.098} C_VEL
LIN {X 0,Y 164.965,Z 616.178,A -85,B 0,C 180,E1 -31803.509,E2 -31803.509} C_VEL
LIN {X 0,Y 172.769,Z 617.262,A -85,B 0,C 180,E1 -31807.461,E2 -31807.461} C_VEL
LIN {X 0,Y 181.298,Z 617.311,A -85,B 0,C 180,E1 -31811.062,E2 -31811.062} C_VEL
LIN {X 0,Y 190.923,Z 616.338,A -85,B 0,C 180,E1 -31814.198,E2 -31814.198} C_VEL
LIN {X 0,Y 201.324,Z 614.293,A -85,B 0,C 180,E1 -31816.945,E2 -31816.945} C_VEL
LIN {X 0,Y 212.381,Z 611.11,A -85,B 0,C 180,E1 -31819.343,E2 -31819.343} C_VEL
LIN {X 0,Y 223.952,Z 606.719,A -85,B 0,C 180,E1 -31821.442,E2 -31821.442} C_VEL
LIN {X 0,Y 222.15,Z 607.373,A -85,B 0,C 180,E1 -31822.029,E2 -31822.029} C_VEL
LIN {X 0,Y 213.205,Z 610.463,A -85,B 0,C 180,E1 -31823.747,E2 -31823.747} C_VEL
LIN {X 0,Y 201.903,Z 613.378,A -85,B 0,C 180,E1 -31826.284,E2 -31826.284} C_VEL
LIN {X 0,Y 191.258,Z 615.061,A -85,B 0,C 180,E1 -31829.155,E2 -31829.155} C_VEL
LIN {X 0,Y 181.427,Z 615.563,A -85,B 0,C 180,E1 -31832.4,E2 -31832.4} C_VEL
LIN {X 0,Y 172.505,Z 614.922,A -85,B 0,C 180,E1 -31836.043,E2 -31836.043} C_VEL
LIN {X 0,Y 164.671,Z 613.164,A -85,B 0,C 180,E1 -31840.105,E2 -31840.105} C_VEL
LIN {X 0,Y 158.141,Z 610.321,A -85,B 0,C 180,E1 -31844.588,E2 -31844.588} C_VEL
LIN {X 0,Y 152.956,Z 606.354,A -85,B 0,C 180,E1 -31849.445,E2 -31849.445} C_VEL
LIN {X 0,Y 149.328,Z 601.235,A -85,B 0,C 180,E1 -31854.617,E2 -31854.617} C_VEL
LIN {X 0,Y 147.108,Z 594.726,A -85,B 0,C 180,E1 -31860.069,E2 -31860.069} C_VEL
LIN {X 0,Y 146.16,Z 586.833,A -85,B 0,C 180,E1 -31865.5,E2 -31865.5} C_VEL
LIN {X 0,Y 146.138,Z 579.566,A -85,B 0,C 180,E1 -31869.657,E2 -31869.657} C_VEL
LIN {X 0,Y 146.375,Z 570.714,A -85,B 0,C 180,E1 -31873.843,E2 -31873.843} C_VEL
LIN {X 0,Y 146.702,Z 560.118,A -85,B 0,C 180,E1 -31877.936,E2 -31877.936} C_VEL
LIN {X 0,Y 147.23,Z 548.433,A -85,B 0,C 180,E1 -31881.636,E2 -31881.636} C_VEL
LIN {X 0,Y 148.004,Z 536.116,A -85,B 0,C 180,E1 -31884.836,E2 -31884.836} C_VEL
LIN {X 0,Y 149.032,Z 522.582,A -85,B 0,C 180,E1 -31887.681,E2 -31887.681} C_VEL
LIN {X 0,Y 150.076,Z 507.808,A -85,B 0,C 180,E1 -31890.115,E2 -31890.115} C_VEL
LIN {X 0,Y 151.089,Z 492.388,A -85,B 0,C 180,E1 -31892.022,E2 -31892.022} C_VEL
LIN {X 0,Y 152.228,Z 471.895,A -85,B 0,C 180,E1 -31893.819,E2 -31893.819} C_VEL
LIN {X 0,Y 156.025,Z 393.465,A -85,B 0,C 180,E1 -31900.121,E2 -31900.121} C_VEL
LIN {X 0,Y 153.94,Z 369.007,A -85,B 0,C 180,E1 -31902.103,E2 -31902.103} C_VEL
LIN {X 0,Y 149.457,Z 348.75,A -85,B 0,C 180,E1 -31903.949,E2 -31903.949} C_VEL
LIN {X 0,Y 149.101,Z 347.084,A -85,B 0,C 180,E1 -31904.532,E2 -31904.532} C_VEL
LIN {X 0,Y 150.065,Z 349.108,A -85,B 0,C 180,E1 -31905.209,E2 -31905.209} C_VEL
LIN {X 0,Y 151.167,Z 349.735,A -85,B 0,C 180,E1 -31905.781,E2 -31905.781} C_VEL
LIN {X 0,Y 153.435,Z 349.144,A -85,B 0,C 180,E1 -31906.775,E2 -31906.775} C_VEL
LIN {X 0,Y 154.591,Z 349.358,A -85,B 0,C 180,E1 -31907.3,E2 -31907.3} C_VEL
LIN {X 0,Y 160.595,Z 358.065,A -85,B 0,C 180,E1 -31910.318,E2 -31910.318} C_VEL
LIN {X 0,Y 167.144,Z 368.562,A -85,B 0,C 180,E1 -31913.265,E2 -31913.265} C_VEL
LIN {X 0,Y 174,Z 381.387,A -85,B 0,C 180,E1 -31916.084,E2 -31916.084} C_VEL
LIN {X 0,Y 179.223,Z 392.82,A -85,B 0,C 180,E1 -31918.104,E2 -31918.104} C_VEL
LIN {X 0,Y 175.092,Z 459.595,A -85,B 0,C 180,E1 -31920.529,E2 -31920.529} C_VEL
LIN {X 0,Y 173.446,Z 474.37,A -85,B 0,C 180,E1 -31921.502,E2 -31921.502} C_VEL
LIN {X 0,Y 171.193,Z 488.658,A -85,B 0,C 180,E1 -31922.917,E2 -31922.917} C_VEL
LIN {X 0,Y 168.207,Z 502.302,A -85,B 0,C 180,E1 -31924.728,E2 -31924.728} C_VEL
LIN {X 0,Y 164.787,Z 514.618,A -85,B 0,C 180,E1 -31926.841,E2 -31926.841} C_VEL
LIN {X 0,Y 161.399,Z 525.851,A -85,B 0,C 180,E1 -31929.347,E2 -31929.347} C_VEL
LIN {X 0,Y 159.086,Z 533.25,A -85,B 0,C 180,E1 -31931.379,E2 -31931.379} C_VEL
LIN {X 0,Y 155.734,Z 542.449,A -85,B 0,C 180,E1 -31934.338,E2 -31934.338} C_VEL
LIN {X 0,Y 152.444,Z 551.632,A -85,B 0,C 180,E1 -31938.061,E2 -31938.061} C_VEL
LIN {X 0,Y 149.551,Z 559.316,A -85,B 0,C 180,E1 -31941.916,E2 -31941.916} C_VEL
LIN {X 0,Y 147.369,Z 566.484,A -85,B 0,C 180,E1 -31946.497,E2 -31946.497} C_VEL
LIN {X 0,Y 145.614,Z 572.487,A -85,B 0,C 180,E1 -31951.371,E2 -31951.371} C_VEL
LIN {X 0,Y 144.343,Z 577.657,A -85,B 0,C 180,E1 -31956.961,E2 -31956.961} C_VEL
LIN {X 0,Y 144.131,Z 580.569,A -85,B 0,C 180,E1 -31961.202,E2 -31961.202} C_VEL
LIN {X 0,Y 144.316,Z 582.034,A -85,B 0,C 180,E1 -31964.037,E2 -31964.037} C_VEL
LIN {X 0,Y 145.271,Z 583.949,A -85,B 0,C 180,E1 -31969.718,E2 -31969.718} C_VEL
LIN {X 0,Y 147.702,Z 584.48,A -85,B 0,C 180,E1 -31975.706,E2 -31975.706} C_VEL
LIN {X 0,Y 150.787,Z 583.683,A -85,B 0,C 180,E1 -31980.721,E2 -31980.721} C_VEL
LIN {X 0,Y 155.282,Z 581.475,A -85,B 0,C 180,E1 -31985.894,E2 -31985.894} C_VEL
LIN {X 0,Y 160.838,Z 577.805,A -85,B 0,C 180,E1 -31990.778,E2 -31990.778} C_VEL
LIN {X 0,Y 165.232,Z 574.389,A -85,B 0,C 180,E1 -31993.891,E2 -31993.891} C_VEL
LIN {X 0,Y 171.106,Z 569.206,A -85,B 0,C 180,E1 -31997.455,E2 -31997.455} C_VEL
LIN {X 0,Y 178.087,Z 562.174,A -85,B 0,C 180,E1 -32001.001,E2 -32001.001} C_VEL
LIN {X 0,Y 185.525,Z 553.502,A -85,B 0,C 180,E1 -32004.254,E2 -32004.254} C_VEL
LIN {X 0,Y 192.829,Z 543.74,A -85,B 0,C 180,E1 -32006.984,E2 -32006.984} C_VEL
LIN {X 0,Y 199.632,Z 533.097,A -85,B 0,C 180,E1 -32009.264,E2 -32009.264} C_VEL
LIN {X 0,Y 205.842,Z 521.531,A -85,B 0,C 180,E1 -32011.179,E2 -32011.179} C_VEL
LIN {X 0,Y 211.097,Z 509.916,A -85,B 0,C 180,E1 -32012.669,E2 -32012.669} C_VEL
LIN {X 0,Y 215.794,Z 496.996,A -85,B 0,C 180,E1 -32013.976,E2 -32013.976} C_VEL
LIN {X 0,Y 219.295,Z 484.848,A -85,B 0,C 180,E1 -32014.913,E2 -32014.913} C_VEL
LIN {X 0,Y 222.365,Z 470.209,A -85,B 0,C 180,E1 -32015.747,E2 -32015.747} C_VEL
LIN {X 0,Y 224.302,Z 456.17,A -85,B 0,C 180,E1 -32016.246,E2 -32016.246} C_VEL
LIN {X 0,Y 226.104,Z 435.3,A -85,B 0,C 180,E1 -32016.795,E2 -32016.795} C_VEL
LIN {X 0,Y 222.082,Z 427.145,A -85,B 0,C 180,E1 -32019.278,E2 -32019.278} C_VEL
LIN {X 0,Y 217.646,Z 418.95,A -85,B 0,C 180,E1 -32022.351,E2 -32022.351} C_VEL
LIN {X 0,Y 214.106,Z 412.975,A -85,B 0,C 180,E1 -32025.161,E2 -32025.161} C_VEL
LIN {X 0,Y 211.545,Z 408.801,A -85,B 0,C 180,E1 -32027.498,E2 -32027.498} C_VEL
LIN {X 0,Y 210.011,Z 406.405,A -85,B 0,C 180,E1 -32029.076,E2 -32029.076} C_VEL
LIN {X 0,Y 207.834,Z 402.829,A -85,B 0,C 180,E1 -32031.704,E2 -32031.704} C_VEL
LIN {X 0,Y 205.609,Z 399.05,A -85,B 0,C 180,E1 -32035.125,E2 -32035.125} C_VEL
LIN {X 0,Y 204.896,Z 398.162,A -85,B 0,C 180,E1 -32036.432,E2 -32036.432} C_VEL
LIN {X 0,Y 203.147,Z 394.788,A -85,B 0,C 180,E1 -32041.56,E2 -32041.56} C_VEL
LIN {X 0,Y 203.033,Z 393.999,A -85,B 0,C 180,E1 -32042.472,E2 -32042.472} C_VEL
LIN {X 0,Y 202.863,Z 394.213,A -85,B 0,C 180,E1 -32047.939,E2 -32047.939} C_VEL
LIN {X 0,Y 204.102,Z 398.018,A -85,B 0,C 180,E1 -32053.31,E2 -32053.31} C_VEL
LIN {X 0,Y 205.976,Z 401.462,A -85,B 0,C 180,E1 -32057.08,E2 -32057.08} C_VEL
LIN {X 0,Y 208.804,Z 407.4,A -85,B 0,C 180,E1 -32061.166,E2 -32061.166} C_VEL
LIN {X 0,Y 211.54,Z 413.074,A -85,B 0,C 180,E1 -32064.19,E2 -32064.19} C_VEL
LIN {X 0,Y 213.808,Z 417.856,A -85,B 0,C 180,E1 -32066.33,E2 -32066.33} C_VEL
LIN {X 0,Y 216.947,Z 424.952,A -85,B 0,C 180,E1 -32068.966,E2 -32068.966} C_VEL
LIN {X 0,Y 220.848,Z 434.617,A -85,B 0,C 180,E1 -32071.872,E2 -32071.872} C_VEL
LIN {X 0,Y 224.934,Z 446.235,A -85,B 0,C 180,E1 -32074.632,E2 -32074.632} C_VEL
LIN {X 0,Y 225.154,Z 446.926,A -85,B 0,C 180,E1 -32074.775,E2 -32074.775} C_VEL
LIN {X 0,Y 222.451,Z 475.425,A -85,B 0,C 180,E1 -32075.519,E2 -32075.519} C_VEL
LIN {X 0,Y 219.916,Z 489.477,A -85,B 0,C 180,E1 -32076.062,E2 -32076.062} C_VEL
LIN {X 0,Y 216.161,Z 503.862,A -85,B 0,C 180,E1 -32076.882,E2 -32076.882} C_VEL
LIN {X 0,Y 211.698,Z 516.562,A -85,B 0,C 180,E1 -32077.828,E2 -32077.828} C_VEL
LIN {X 0,Y 206.282,Z 528.961,A -85,B 0,C 180,E1 -32079.046,E2 -32079.046} C_VEL
LIN {X 0,Y 200.485,Z 540.295,A -85,B 0,C 180,E1 -32080.554,E2 -32080.554} C_VEL
LIN {X 0,Y 194.148,Z 550.75,A -85,B 0,C 180,E1 -32082.312,E2 -32082.312} C_VEL
LIN {X 0,Y 187.034,Z 561.162,A -85,B 0,C 180,E1 -32084.647,E2 -32084.647} C_VEL
LIN {X 0,Y 179.236,Z 571.088,A -85,B 0,C 180,E1 -32087.622,E2 -32087.622} C_VEL
LIN {X 0,Y 173.237,Z 577.734,A -85,B 0,C 180,E1 -32090.195,E2 -32090.195} C_VEL
LIN {X 0,Y 166.173,Z 584.845,A -85,B 0,C 180,E1 -32093.842,E2 -32093.842} C_VEL
LIN {X 0,Y 159.432,Z 590.876,A -85,B 0,C 180,E1 -32098.191,E2 -32098.191} C_VEL
LIN {X 0,Y 153.893,Z 595.376,A -85,B 0,C 180,E1 -32102.933,E2 -32102.933} C_VEL
LIN {X 0,Y 149.507,Z 598.47,A -85,B 0,C 180,E1 -32107.995,E2 -32107.995} C_VEL
LIN {X 0,Y 146.356,Z 600.241,A -85,B 0,C 180,E1 -32113.32,E2 -32113.32} C_VEL
LIN {X 0,Y 144.559,Z 600.73,A -85,B 0,C 180,E1 -32118.832,E2 -32118.832} C_VEL
LIN {X 0,Y 144.098,Z 599.936,A -85,B 0,C 180,E1 -32124.428,E2 -32124.428} C_VEL
LIN {X 0,Y 145.02,Z 597.843,A -85,B 0,C 180,E1 -32130.007,E2 -32130.007} C_VEL
LIN {X 0,Y 146.181,Z 595.15,A -85,B 0,C 180,E1 -32134.346,E2 -32134.346} C_VEL
LIN {X 0,Y 147.2,Z 593.016,A -85,B 0,C 180,E1 -32137.182,E2 -32137.182} C_VEL
LIN {X 0,Y 147.264,Z 599.637,A -85,B 0,C 180,E1 -32142.366,E2 -32142.366} C_VEL
LIN {X 0,Y 148.083,Z 603.176,A -85,B 0,C 180,E1 -32145.585,E2 -32145.585} C_VEL
LIN {X 0,Y 148.303,Z 605.106,A -85,B 0,C 180,E1 -32147.742,E2 -32147.742} C_VEL
LIN {X 0,Y 147.603,Z 607.479,A -85,B 0,C 180,E1 -32151.46,E2 -32151.46} C_VEL
LIN {X 0,Y 147.473,Z 609.12,A -85,B 0,C 180,E1 -32154.481,E2 -32154.481} C_VEL
LIN {X 0,Y 148.406,Z 610.477,A -85,B 0,C 180,E1 -32156.686,E2 -32156.686} C_VEL
LIN {X 0,Y 149.007,Z 610.894,A -85,B 0,C 180,E1 -32157.384,E2 -32157.384} C_VEL
LIN {X 0,Y 155.583,Z 614.246,A -85,B 0,C 180,E1 -32162.707,E2 -32162.707} C_VEL
LIN {X 0,Y 162.981,Z 616.199,A -85,B 0,C 180,E1 -32166.997,E2 -32166.997} C_VEL
LIN {X 0,Y 171.543,Z 617.122,A -85,B 0,C 180,E1 -32170.798,E2 -32170.798} C_VEL
LIN {X 0,Y 176.007,Z 617.187,A -85,B 0,C 180,E1 -32172.58,E2 -32172.58} C_VEL
LIN {X 0,Y 185.901,Z 616.579,A -85,B 0,C 180,E1 -32175.723,E2 -32175.723} C_VEL
LIN {X 0,Y 196.555,Z 614.931,A -85,B 0,C 180,E1 -32178.455,E2 -32178.455} C_VEL
LIN {X 0,Y 209.651,Z 611.657,A -85,B 0,C 180,E1 -32181.154,E2 -32181.154} C_VEL
LIN {X 0,Y 210.796,Z 611.274,A -85,B 0,C 180,E1 -32181.887,E2 -32181.887} C_VEL
LIN {X 0,Y 197.224,Z 614.282,A -85,B 0,C 180,E1 -32184.778,E2 -32184.778} C_VEL
LIN {X 0,Y 185.028,Z 615.648,A -85,B 0,C 180,E1 -32187.995,E2 -32187.995} C_VEL
LIN {X 0,Y 175.03,Z 615.636,A -85,B 0,C 180,E1 -32191.3,E2 -32191.3} C_VEL
LIN {X 0,Y 165.913,Z 614.504,A -85,B 0,C 180,E1 -32195.028,E2 -32195.028} C_VEL
LIN {X 0,Y 156.366,Z 611.665,A -85,B 0,C 180,E1 -32200.185,E2 -32200.185} C_VEL
LIN {X 0,Y 149.873,Z 607.986,A -85,B 0,C 180,E1 -32205.105,E2 -32205.105} C_VEL
LIN {X 0,Y 145.025,Z 603.274,A -85,B 0,C 180,E1 -32210.268,E2 -32210.268} C_VEL
LIN {X 0,Y 141.775,Z 597.382,A -85,B 0,C 180,E1 -32215.75,E2 -32215.75} C_VEL
LIN {X 0,Y 140.117,Z 591.005,A -85,B 0,C 180,E1 -32220.79,E2 -32220.79} C_VEL
LIN {X 0,Y 139.461,Z 582.365,A -85,B 0,C 180,E1 -32226.489,E2 -32226.489} C_VEL
LIN {X 0,Y 139.525,Z 574.267,A -85,B 0,C 180,E1 -32230.851,E2 -32230.851} C_VEL
LIN {X 0,Y 139.695,Z 566.145,A -85,B 0,C 180,E1 -32234.519,E2 -32234.519} C_VEL
LIN {X 0,Y 139.981,Z 555.705,A -85,B 0,C 180,E1 -32238.429,E2 -32238.429} C_VEL
LIN {X 0,Y 140.564,Z 543.02,A -85,B 0,C 180,E1 -32242.331,E2 -32242.331} C_VEL
LIN {X 0,Y 141.45,Z 529.648,A -85,B 0,C 180,E1 -32245.676,E2 -32245.676} C_VEL
LIN {X 0,Y 142.424,Z 516.002,A -85,B 0,C 180,E1 -32248.368,E2 -32248.368} C_VEL
LIN {X 0,Y 143.329,Z 502.482,A -85,B 0,C 180,E1 -32250.466,E2 -32250.466} C_VEL
LIN {X 0,Y 144.341,Z 488.12,A -85,B 0,C 180,E1 -32252.16,E2 -32252.16} C_VEL
LIN {X 0,Y 146.257,Z 444.323,A -85,B 0,C 180,E1 -32256.025,E2 -32256.025} C_VEL
LIN {X 0,Y 148.926,Z 393.733,A -85,B 0,C 180,E1 -32260.249,E2 -32260.249} C_VEL
LIN {X 0,Y 146.995,Z 370.374,A -85,B 0,C 180,E1 -32262.239,E2 -32262.239} C_VEL
LIN {X 0,Y 144.623,Z 359.616,A -85,B 0,C 180,E1 -32263.274,E2 -32263.274} C_VEL
LIN {X 0,Y 145.589,Z 361.795,A -85,B 0,C 180,E1 -32263.963,E2 -32263.963} C_VEL
LIN {X 0,Y 146.812,Z 362.127,A -85,B 0,C 180,E1 -32264.616,E2 -32264.616} C_VEL
LIN {X 0,Y 148.114,Z 361.102,A -85,B 0,C 180,E1 -32265.183,E2 -32265.183} C_VEL
LIN {X 0,Y 149.933,Z 357.959,A -85,B 0,C 180,E1 -32265.818,E2 -32265.818} C_VEL
LIN {X 0,Y 150.43,Z 356.766,A -85,B 0,C 180,E1 -32265.962,E2 -32265.962} C_VEL
LIN {X 0,Y 152.429,Z 356.845,A -85,B 0,C 180,E1 -32266.883,E2 -32266.883} C_VEL
LIN {X 0,Y 154.952,Z 360.461,A -85,B 0,C 180,E1 -32268.234,E2 -32268.234} C_VEL
LIN {X 0,Y 160.624,Z 369.214,A -85,B 0,C 180,E1 -32271.042,E2 -32271.042} C_VEL
LIN {X 0,Y 166.777,Z 380.359,A -85,B 0,C 180,E1 -32273.836,E2 -32273.836} C_VEL
LIN {X 0,Y 172.174,Z 391.693,A -85,B 0,C 180,E1 -32276.119,E2 -32276.119} C_VEL
LIN {X 0,Y 173.589,Z 394.919,A -85,B 0,C 180,E1 -32276.696,E2 -32276.696} C_VEL
LIN {X 0,Y 169.408,Z 460.217,A -85,B 0,C 180,E1 -32279.13,E2 -32279.13} C_VEL
LIN {X 0,Y 167.73,Z 474.599,A -85,B 0,C 180,E1 -32280.092,E2 -32280.092} C_VEL
LIN {X 0,Y 165.395,Z 488.925,A -85,B 0,C 180,E1 -32281.541,E2 -32281.541} C_VEL
LIN {X 0,Y 162.274,Z 502.603,A -85,B 0,C 180,E1 -32283.389,E2 -32283.389} C_VEL
LIN {X 0,Y 158.715,Z 514.939,A -85,B 0,C 180,E1 -32285.554,E2 -32285.554} C_VEL
LIN {X 0,Y 155.172,Z 526.188,A -85,B 0,C 180,E1 -32288.13,E2 -32288.13} C_VEL
LIN {X 0,Y 152.359,Z 534.579,A -85,B 0,C 180,E1 -32290.524,E2 -32290.524} C_VEL
LIN {X 0,Y 148.286,Z 545.249,A -85,B 0,C 180,E1 -32294.234,E2 -32294.234} C_VEL
LIN {X 0,Y 144.959,Z 554.036,A -85,B 0,C 180,E1 -32298.143,E2 -32298.143} C_VEL
LIN {X 0,Y 142.173,Z 561.36,A -85,B 0,C 180,E1 -32302.207,E2 -32302.207} C_VEL
LIN {X 0,Y 139.944,Z 568.349,A -85,B 0,C 180,E1 -32307.124,E2 -32307.124} C_VEL
LIN {X 0,Y 138.446,Z 573.239,A -85,B 0,C 180,E1 -32311.442,E2 -32311.442} C_VEL
LIN {X 0,Y 137.201,Z 578.328,A -85,B 0,C 180,E1 -32317.325,E2 -32317.325} C_VEL
LIN {X 0,Y 137.062,Z 581.161,A -85,B 0,C 180,E1 -32321.788,E2 -32321.788} C_VEL
LIN {X 0,Y 137.284,Z 582.59,A -85,B 0,C 180,E1 -32324.772,E2 -32324.772} C_VEL
LIN {X 0,Y 138.431,Z 584.431,A -85,B 0,C 180,E1 -32330.736,E2 -32330.736} C_VEL
LIN {X 0,Y 140.917,Z 584.902,A -85,B 0,C 180,E1 -32336.566,E2 -32336.566} C_VEL
LIN {X 0,Y 144.531,Z 584.014,A -85,B 0,C 180,E1 -32342.206,E2 -32342.206} C_VEL
LIN {X 0,Y 149.395,Z 581.727,A -85,B 0,C 180,E1 -32347.545,E2 -32347.545} C_VEL
LIN {X 0,Y 155.369,Z 577.977,A -85,B 0,C 180,E1 -32352.541,E2 -32352.541} C_VEL
LIN {X 0,Y 160.646,Z 573.999,A -85,B 0,C 180,E1 -32356.088,E2 -32356.088} C_VEL
LIN {X 0,Y 166.257,Z 569.207,A -85,B 0,C 180,E1 -32359.308,E2 -32359.308} C_VEL
LIN {X 0,Y 172.895,Z 562.783,A -85,B 0,C 180,E1 -32362.577,E2 -32362.577} C_VEL
LIN {X 0,Y 180.203,Z 554.668,A -85,B 0,C 180,E1 -32365.677,E2 -32365.677} C_VEL
LIN {X 0,Y 187.449,Z 545.431,A -85,B 0,C 180,E1 -32368.336,E2 -32368.336} C_VEL
LIN {X 0,Y 193.479,Z 536.601,A -85,B 0,C 180,E1 -32370.315,E2 -32370.315} C_VEL
LIN {X 0,Y 199.829,Z 525.748,A -85,B 0,C 180,E1 -32372.247,E2 -32372.247} C_VEL
LIN {X 0,Y 205.306,Z 514.709,A -85,B 0,C 180,E1 -32373.783,E2 -32373.783} C_VEL
LIN {X 0,Y 210.356,Z 502.365,A -85,B 0,C 180,E1 -32375.131,E2 -32375.131} C_VEL
LIN {X 0,Y 214.35,Z 490.036,A -85,B 0,C 180,E1 -32376.188,E2 -32376.188} C_VEL
LIN {X 0,Y 217.91,Z 475.566,A -85,B 0,C 180,E1 -32377.099,E2 -32377.099} C_VEL
LIN {X 0,Y 220.299,Z 461.263,A -85,B 0,C 180,E1 -32377.702,E2 -32377.702} C_VEL
LIN {X 0,Y 222.37,Z 438.552,A -85,B 0,C 180,E1 -32378.338,E2 -32378.338} C_VEL
LIN {X 0,Y 217.828,Z 429.35,A -85,B 0,C 180,E1 -32381.416,E2 -32381.416} C_VEL
LIN {X 0,Y 213.693,Z 421.684,A -85,B 0,C 180,E1 -32384.646,E2 -32384.646} C_VEL
LIN {X 0,Y 210.561,Z 416.369,A -85,B 0,C 180,E1 -32387.493,E2 -32387.493} C_VEL
LIN {X 0,Y 208.717,Z 413.27,A -85,B 0,C 180,E1 -32389.451,E2 -32389.451} C_VEL
LIN {X 0,Y 206.529,Z 409.578,A -85,B 0,C 180,E1 -32392.203,E2 -32392.203} C_VEL
LIN {X 0,Y 204.402,Z 405.747,A -85,B 0,C 180,E1 -32395.679,E2 -32395.679} C_VEL
LIN {X 0,Y 202.251,Z 401.986,A -85,B 0,C 180,E1 -32401.566,E2 -32401.566} C_VEL
LIN {X 0,Y 202.123,Z 401.124,A -85,B 0,C 180,E1 -32402.6,E2 -32402.6} C_VEL
LIN {X 0,Y 201.936,Z 401.177,A -85,B 0,C 180,E1 -32407.474,E2 -32407.474} C_VEL
LIN {X 0,Y 203.025,Z 404.828,A -85,B 0,C 180,E1 -32412.832,E2 -32412.832} C_VEL
LIN {X 0,Y 204.715,Z 408.126,A -85,B 0,C 180,E1 -32416.495,E2 -32416.495} C_VEL
LIN {X 0,Y 207.365,Z 414.04,A -85,B 0,C 180,E1 -32420.579,E2 -32420.579} C_VEL
LIN {X 0,Y 209.841,Z 419.511,A -85,B 0,C 180,E1 -32423.498,E2 -32423.498} C_VEL
LIN {X 0,Y 212.226,Z 424.826,A -85,B 0,C 180,E1 -32425.867,E2 -32425.867} C_VEL
LIN {X 0,Y 215.721,Z 433.335,A -85,B 0,C 180,E1 -32428.911,E2 -32428.911} C_VEL
LIN {X 0,Y 219.215,Z 442.859,A -85,B 0,C 180,E1 -32431.616,E2 -32431.616} C_VEL
LIN {X 0,Y 221.481,Z 449.678,A -85,B 0,C 180,E1 -32433.242,E2 -32433.242} C_VEL
LIN {X 0,Y 218.976,Z 475.185,A -85,B 0,C 180,E1 -32433.916,E2 -32433.916} C_VEL
LIN {X 0,Y 216.204,Z 489.918,A -85,B 0,C 180,E1 -32434.48,E2 -32434.48} C_VEL
LIN {X 0,Y 212.358,Z 504.105,A -85,B 0,C 180,E1 -32435.288,E2 -32435.288} C_VEL
LIN {X 0,Y 207.431,Z 517.543,A -85,B 0,C 180,E1 -32436.283,E2 -32436.283} C_VEL
LIN {X 0,Y 201.906,Z 529.671,A -85,B 0,C 180,E1 -32437.489,E2 -32437.489} C_VEL
LIN {X 0,Y 195.296,Z 541.931,A -85,B 0,C 180,E1 -32439.15,E2 -32439.15} C_VEL
LIN {X 0,Y 188.227,Z 552.946,A -85,B 0,C 180,E1 -32441.11,E2 -32441.11} C_VEL
LIN {X 0,Y 180.944,Z 562.877,A -85,B 0,C 180,E1 -32443.471,E2 -32443.471} C_VEL
LIN {X 0,Y 172.932,Z 572.391,A -85,B 0,C 180,E1 -32446.492,E2 -32446.492} C_VEL
LIN {X 0,Y 165.252,Z 580.27,A -85,B 0,C 180,E1 -32449.851,E2 -32449.851} C_VEL
LIN {X 0,Y 158.605,Z 586.373,A -85,B 0,C 180,E1 -32453.41,E2 -32453.41} C_VEL
LIN {X 0,Y 151.852,Z 591.961,A -85,B 0,C 180,E1 -32457.972,E2 -32457.972} C_VEL
LIN {X 0,Y 147.559,Z 595.129,A -85,B 0,C 180,E1 -32461.669,E2 -32461.669} C_VEL
LIN {X 0,Y 142.91,Z 598.16,A -85,B 0,C 180,E1 -32466.922,E2 -32466.922} C_VEL
LIN {X 0,Y 139.475,Z 599.892,A -85,B 0,C 180,E1 -32472.589,E2 -32472.589} C_VEL
LIN {X 0,Y 137.569,Z 600.299,A -85,B 0,C 180,E1 -32478.256,E2 -32478.256} C_VEL
LIN {X 0,Y 137.01,Z 599.444,A -85,B 0,C 180,E1 -32484.139,E2 -32484.139} C_VEL
LIN {X 0,Y 137.92,Z 597.291,A -85,B 0,C 180,E1 -32490.007,E2 -32490.007} C_VEL
LIN {X 0,Y 138.699,Z 595.694,A -85,B 0,C 180,E1 -32492.902,E2 -32492.902} C_VEL
LIN {X 0,Y 140.592,Z 591.649,A -85,B 0,C 180,E1 -32498.332,E2 -32498.332} C_VEL
LIN {X 0,Y 140.988,Z 599.082,A -85,B 0,C 180,E1 -32504.39,E2 -32504.39} C_VEL
LIN {X 0,Y 143.167,Z 604.835,A -85,B 0,C 180,E1 -32510.035,E2 -32510.035} C_VEL
LIN {X 0,Y 147.116,Z 609.436,A -85,B 0,C 180,E1 -32515.38,E2 -32515.38} C_VEL
LIN {X 0,Y 149.007,Z 610.894,A -85,B 0,C 180,E1 -32517.384,E2 -32517.384} C_VEL
LIN {X 0,Y 150.581,Z 612.211,A -85,B 0,C 180,E1 -32519.508,E2 -32519.508} C_VEL
LIN {X 0,Y 152.173,Z 613.712,A -85,B 0,C 180,E1 -32523.177,E2 -32523.177} C_VEL
LIN {X 0,Y 154.663,Z 614.77,A -85,B 0,C 180,E1 -32526.726,E2 -32526.726} C_VEL
LIN {X 0,Y 157.538,Z 615.391,A -85,B 0,C 180,E1 -32528.593,E2 -32528.593} C_VEL
LIN {X 0,Y 166.241,Z 616.664,A -85,B 0,C 180,E1 -32532.395,E2 -32532.395} C_VEL
LIN {X 0,Y 170.851,Z 616.933,A -85,B 0,C 180,E1 -32534.19,E2 -32534.19} C_VEL
LIN {X 0,Y 181.017,Z 616.717,A -85,B 0,C 180,E1 -32537.332,E2 -32537.332} C_VEL
LIN {X 0,Y 191.929,Z 615.459,A -85,B 0,C 180,E1 -32540.038,E2 -32540.038} C_VEL
LIN {X 0,Y 197.667,Z 614.429,A -85,B 0,C 180,E1 -32541.229,E2 -32541.229} C_VEL
LIN {X 0,Y 198.676,Z 614.194,A -85,B 0,C 180,E1 -32541.895,E2 -32541.895} C_VEL
LIN {X 0,Y 189.947,Z 615.401,A -85,B 0,C 180,E1 -32543.842,E2 -32543.842} C_VEL
LIN {X 0,Y 178.897,Z 616.007,A -85,B 0,C 180,E1 -32546.76,E2 -32546.76} C_VEL
LIN {X 0,Y 168.687,Z 615.484,A -85,B 0,C 180,E1 -32550.114,E2 -32550.114} C_VEL
LIN {X 0,Y 159.395,Z 613.866,A -85,B 0,C 180,E1 -32553.932,E2 -32553.932} C_VEL
LIN {X 0,Y 150.027,Z 610.6,A -85,B 0,C 180,E1 -32559.044,E2 -32559.044} C_VEL
LIN {X 0,Y 143.088,Z 606.294,A -85,B 0,C 180,E1 -32564.381,E2 -32564.381} C_VEL
LIN {X 0,Y 138.189,Z 601.13,A -85,B 0,C 180,E1 -32569.781,E2 -32569.781} C_VEL
LIN {X 0,Y 134.982,Z 594.786,A -85,B 0,C 180,E1 -32575.536,E2 -32575.536} C_VEL
LIN {X 0,Y 133.168,Z 586.497,A -85,B 0,C 180,E1 -32581.847,E2 -32581.847} C_VEL
LIN {X 0,Y 132.835,Z 578.684,A -85,B 0,C 180,E1 -32586.814,E2 -32586.814} C_VEL
LIN {X 0,Y 132.879,Z 569.97,A -85,B 0,C 180,E1 -32591.401,E2 -32591.401} C_VEL
LIN {X 0,Y 133.014,Z 561.067,A -85,B 0,C 180,E1 -32595.266,E2 -32595.266} C_VEL
LIN {X 0,Y 133.28,Z 551.123,A -85,B 0,C 180,E1 -32598.899,E2 -32598.899} C_VEL
LIN {X 0,Y 133.817,Z 539.997,A -85,B 0,C 180,E1 -32602.302,E2 -32602.302} C_VEL
LIN {X 0,Y 134.726,Z 525.869,A -85,B 0,C 180,E1 -32605.812,E2 -32605.812} C_VEL
LIN {X 0,Y 135.617,Z 512.84,A -85,B 0,C 180,E1 -32608.391,E2 -32608.391} C_VEL
LIN {X 0,Y 136.604,Z 498.138,A -85,B 0,C 180,E1 -32610.645,E2 -32610.645} C_VEL
LIN {X 0,Y 137.741,Z 480.334,A -85,B 0,C 180,E1 -32612.596,E2 -32612.596} C_VEL
LIN {X 0,Y 141.83,Z 394.088,A -85,B 0,C 180,E1 -32620.363,E2 -32620.363} C_VEL
LIN {X 0,Y 140.286,Z 374.597,A -85,B 0,C 180,E1 -32622.136,E2 -32622.136} C_VEL
LIN {X 0,Y 140.893,Z 377.173,A -85,B 0,C 180,E1 -32622.706,E2 -32622.706} C_VEL
LIN {X 0,Y 141.59,Z 377.912,A -85,B 0,C 180,E1 -32623.157,E2 -32623.157} C_VEL
LIN {X 0,Y 142.908,Z 377.381,A -85,B 0,C 180,E1 -32623.827,E2 -32623.827} C_VEL
LIN {X 0,Y 144.604,Z 374.73,A -85,B 0,C 180,E1 -32624.498,E2 -32624.498} C_VEL
LIN {X 0,Y 146.856,Z 369.175,A -85,B 0,C 180,E1 -32625.192,E2 -32625.192} C_VEL
LIN {X 0,Y 149.497,Z 367.549,A -85,B 0,C 180,E1 -32626.334,E2 -32626.334} C_VEL
LIN {X 0,Y 150.895,Z 365.984,A -85,B 0,C 180,E1 -32626.86,E2 -32626.86} C_VEL
LIN {X 0,Y 151.676,Z 366.184,A -85,B 0,C 180,E1 -32627.225,E2 -32627.225} C_VEL
LIN {X 0,Y 156.884,Z 374.567,A -85,B 0,C 180,E1 -32629.973,E2 -32629.973} C_VEL
LIN {X 0,Y 162.493,Z 384.947,A -85,B 0,C 180,E1 -32632.686,E2 -32632.686} C_VEL
LIN {X 0,Y 167.969,Z 396.847,A -85,B 0,C 180,E1 -32635.157,E2 -32635.157} C_VEL
LIN {X 0,Y 168.128,Z 398.746,A -85,B 0,C 180,E1 -32635.313,E2 -32635.313} C_VEL
LIN {X 0,Y 163.891,Z 460.282,A -85,B 0,C 180,E1 -32637.605,E2 -32637.605} C_VEL
LIN {X 0,Y 162.124,Z 474.887,A -85,B 0,C 180,E1 -32638.593,E2 -32638.593} C_VEL
LIN {X 0,Y 159.699,Z 489.188,A -85,B 0,C 180,E1 -32640.066,E2 -32640.066} C_VEL
LIN {X 0,Y 156.436,Z 502.902,A -85,B 0,C 180,E1 -32641.95,E2 -32641.95} C_VEL
LIN {X 0,Y 152.73,Z 515.26,A -85,B 0,C 180,E1 -32644.164,E2 -32644.164} C_VEL
LIN {X 0,Y 149.02,Z 526.526,A -85,B 0,C 180,E1 -32646.811,E2 -32646.811} C_VEL
LIN {X 0,Y 146.476,Z 533.947,A -85,B 0,C 180,E1 -32648.976,E2 -32648.976} C_VEL
LIN {X 0,Y 142.776,Z 543.171,A -85,B 0,C 180,E1 -32652.138,E2 -32652.138} C_VEL
LIN {X 0,Y 139.137,Z 552.371,A -85,B 0,C 180,E1 -32656.158,E2 -32656.158} C_VEL
LIN {X 0,Y 135.944,Z 560.069,A -85,B 0,C 180,E1 -32660.353,E2 -32660.353} C_VEL
LIN {X 0,Y 133.533,Z 567.156,A -85,B 0,C 180,E1 -32665.302,E2 -32665.302} C_VEL
LIN {X 0,Y 131.754,Z 572.52,A -85,B 0,C 180,E1 -32669.993,E2 -32669.993} C_VEL
LIN {X 0,Y 130.527,Z 576.69,A -85,B 0,C 180,E1 -32674.609,E2 -32674.609} C_VEL
LIN {X 0,Y 129.978,Z 580.013,A -85,B 0,C 180,E1 -32679.296,E2 -32679.296} C_VEL
LIN {X 0,Y 130.277,Z 583.147,A -85,B 0,C 180,E1 -32685.587,E2 -32685.587} C_VEL
LIN {X 0,Y 131.641,Z 584.912,A -85,B 0,C 180,E1 -32691.859,E2 -32691.859} C_VEL
LIN {X 0,Y 134.419,Z 585.309,A -85,B 0,C 180,E1 -32697.96,E2 -32697.96} C_VEL
LIN {X 0,Y 138.384,Z 584.346,A -85,B 0,C 180,E1 -32703.824,E2 -32703.824} C_VEL
LIN {X 0,Y 143.644,Z 581.985,A -85,B 0,C 180,E1 -32709.33,E2 -32709.33} C_VEL
LIN {X 0,Y 150.059,Z 578.134,A -85,B 0,C 180,E1 -32714.431,E2 -32714.431} C_VEL
LIN {X 0,Y 157.513,Z 572.625,A -85,B 0,C 180,E1 -32719.1,E2 -32719.1} C_VEL
LIN {X 0,Y 164.782,Z 566.335,A -85,B 0,C 180,E1 -32722.835,E2 -32722.835} C_VEL
LIN {X 0,Y 172.655,Z 558.428,A -85,B 0,C 180,E1 -32726.258,E2 -32726.258} C_VEL
LIN {X 0,Y 179.829,Z 550.1,A -85,B 0,C 180,E1 -32728.96,E2 -32728.96} C_VEL
LIN {X 0,Y 187.389,Z 540.001,A -85,B 0,C 180,E1 -32731.438,E2 -32731.438} C_VEL
LIN {X 0,Y 193.919,Z 529.781,A -85,B 0,C 180,E1 -32733.365,E2 -32733.365} C_VEL
LIN {X 0,Y 199.704,Z 519.029,A -85,B 0,C 180,E1 -32734.985,E2 -32734.985} C_VEL
LIN {X 0,Y 205.322,Z 506.524,A -85,B 0,C 180,E1 -32736.452,E2 -32736.452} C_VEL
LIN {X 0,Y 210.103,Z 492.973,A -85,B 0,C 180,E1 -32737.674,E2 -32737.674} C_VEL
LIN {X 0,Y 213.925,Z 478.776,A -85,B 0,C 180,E1 -32738.589,E2 -32738.589} C_VEL
LIN {X 0,Y 216.531,Z 464.749,A -85,B 0,C 180,E1 -32739.23,E2 -32739.23} C_VEL
LIN {X 0,Y 218.61,Z 445.249,A -85,B 0,C 180,E1 -32739.781,E2 -32739.781} C_VEL
LIN {X 0,Y 218.802,Z 442.037,A -85,B 0,C 180,E1 -32739.915,E2 -32739.915} C_VEL
LIN {X 0,Y 214.727,Z 433.599,A -85,B 0,C 180,E1 -32742.928,E2 -32742.928} C_VEL
LIN {X 0,Y 211.167,Z 426.796,A -85,B 0,C 180,E1 -32745.963,E2 -32745.963} C_VEL
LIN {X 0,Y 207.66,Z 420.441,A -85,B 0,C 180,E1 -32749.576,E2 -32749.576} C_VEL
LIN {X 0,Y 205.13,Z 416.16,A -85,B 0,C 180,E1 -32752.867,E2 -32752.867} C_VEL
LIN {X 0,Y 203.084,Z 412.289,A -85,B 0,C 180,E1 -32756.497,E2 -32756.497} C_VEL
LIN {X 0,Y 201.377,Z 409.305,A -85,B 0,C 180,E1 -32761.433,E2 -32761.433} C_VEL
LIN {X 0,Y 201.152,Z 408.063,A -85,B 0,C 180,E1 -32763.23,E2 -32763.23} C_VEL
LIN {X 0,Y 201.06,Z 408.271,A -85,B 0,C 180,E1 -32767.507,E2 -32767.507} C_VEL
LIN {X 0,Y 202.016,Z 411.775,A -85,B 0,C 180,E1 -32772.516,E2 -32772.516} C_VEL
LIN {X 0,Y 203.556,Z 415.024,A -85,B 0,C 180,E1 -32776.07,E2 -32776.07} C_VEL
LIN {X 0,Y 205.877,Z 420.556,A -85,B 0,C 180,E1 -32779.891,E2 -32779.891} C_VEL
LIN {X 0,Y 208.094,Z 425.788,A -85,B 0,C 180,E1 -32782.708,E2 -32782.708} C_VEL
LIN {X 0,Y 210.268,Z 430.927,A -85,B 0,C 180,E1 -32785.018,E2 -32785.018} C_VEL
LIN {X 0,Y 213.459,Z 439.137,A -85,B 0,C 180,E1 -32787.991,E2 -32787.991} C_VEL
LIN {X 0,Y 216.617,Z 448.318,A -85,B 0,C 180,E1 -32790.616,E2 -32790.616} C_VEL
LIN {X 0,Y 217.973,Z 452.576,A -85,B 0,C 180,E1 -32791.67,E2 -32791.67} C_VEL
LIN {X 0,Y 215.634,Z 475.167,A -85,B 0,C 180,E1 -32792.264,E2 -32792.264} C_VEL
LIN {X 0,Y 212.806,Z 489.78,A -85,B 0,C 180,E1 -32792.82,E2 -32792.82} C_VEL
LIN {X 0,Y 209.074,Z 503.23,A -85,B 0,C 180,E1 -32793.564,E2 -32793.564} C_VEL
LIN {X 0,Y 204.034,Z 516.767,A -85,B 0,C 180,E1 -32794.531,E2 -32794.531} C_VEL
LIN {X 0,Y 198.378,Z 528.963,A -85,B 0,C 180,E1 -32795.709,E2 -32795.709} C_VEL
LIN {X 0,Y 192.265,Z 540.15,A -85,B 0,C 180,E1 -32797.172,E2 -32797.172} C_VEL
LIN {X 0,Y 184.917,Z 551.451,A -85,B 0,C 180,E1 -32799.067,E2 -32799.067} C_VEL
LIN {X 0,Y 177.354,Z 561.566,A -85,B 0,C 180,E1 -32801.385,E2 -32801.385} C_VEL
LIN {X 0,Y 170.151,Z 569.997,A -85,B 0,C 180,E1 -32803.921,E2 -32803.921} C_VEL
LIN {X 0,Y 162.099,Z 578.179,A -85,B 0,C 180,E1 -32807.198,E2 -32807.198} C_VEL
LIN {X 0,Y 154.927,Z 584.65,A -85,B 0,C 180,E1 -32810.74,E2 -32810.74} C_VEL
LIN {X 0,Y 147.544,Z 590.527,A -85,B 0,C 180,E1 -32815.281,E2 -32815.281} C_VEL
LIN {X 0,Y 141.307,Z 594.886,A -85,B 0,C 180,E1 -32820.293,E2 -32820.293} C_VEL
LIN {X 0,Y 136.386,Z 597.852,A -85,B 0,C 180,E1 -32825.749,E2 -32825.749} C_VEL
LIN {X 0,Y 132.479,Z 599.605,A -85,B 0,C 180,E1 -32832.119,E2 -32832.119} C_VEL
LIN {X 0,Y 130.596,Z 599.867,A -85,B 0,C 180,E1 -32837.62,E2 -32837.62} C_VEL
LIN {X 0,Y 129.928,Z 598.952,A -85,B 0,C 180,E1 -32843.818,E2 -32843.818} C_VEL
LIN {X 0,Y 130.828,Z 596.739,A -85,B 0,C 180,E1 -32850.007,E2 -32850.007} C_VEL
LIN {X 0,Y 132.031,Z 594.134,A -85,B 0,C 180,E1 -32854.572,E2 -32854.572} C_VEL
LIN {X 0,Y 134.029,Z 590.305,A -85,B 0,C 180,E1 -32859.691,E2 -32859.691} C_VEL
LIN {X 0,Y 134.486,Z 596.835,A -85,B 0,C 180,E1 -32865.102,E2 -32865.102} C_VEL
LIN {X 0,Y 136.766,Z 602.917,A -85,B 0,C 180,E1 -32871.016,E2 -32871.016} C_VEL
LIN {X 0,Y 140.91,Z 607.841,A -85,B 0,C 180,E1 -32876.583,E2 -32876.583} C_VEL
LIN {X 0,Y 146.413,Z 611.6,A -85,B 0,C 180,E1 -32881.759,E2 -32881.759} C_VEL
LIN {X 0,Y 153.444,Z 614.363,A -85,B 0,C 180,E1 -32886.408,E2 -32886.408} C_VEL
LIN {X 0,Y 157.538,Z 615.391,A -85,B 0,C 180,E1 -32888.593,E2 -32888.593} C_VEL
LIN {X 0,Y 160.628,Z 616.001,A -85,B 0,C 180,E1 -32890.392,E2 -32890.392} C_VEL
LIN {X 0,Y 164.581,Z 616.498,A -85,B 0,C 180,E1 -32893.59,E2 -32893.59} C_VEL
LIN {X 0,Y 169.104,Z 616.707,A -85,B 0,C 180,E1 -32896.611,E2 -32896.611} C_VEL
LIN {X 0,Y 172.968,Z 616.698,A -85,B 0,C 180,E1 -32898.097,E2 -32898.097} C_VEL
LIN {X 0,Y 181.78,Z 616.399,A -85,B 0,C 180,E1 -32900.42,E2 -32900.42} C_VEL
LIN {X 0,Y 187.349,Z 615.863,A -85,B 0,C 180,E1 -32901.74,E2 -32901.74} C_VEL
LIN {X 0,Y 178.371,Z 616.231,A -85,B 0,C 180,E1 -32903.911,E2 -32903.911} C_VEL
LIN {X 0,Y 165.992,Z 615.589,A -85,B 0,C 180,E1 -32907.569,E2 -32907.569} C_VEL
LIN {X 0,Y 157.56,Z 614.184,A -85,B 0,C 180,E1 -32910.724,E2 -32910.724} C_VEL
LIN {X 0,Y 148.685,Z 611.562,A -85,B 0,C 180,E1 -32914.913,E2 -32914.913} C_VEL
LIN {X 0,Y 141.099,Z 607.885,A -85,B 0,C 180,E1 -32919.666,E2 -32919.666} C_VEL
LIN {X 0,Y 134.993,Z 603.117,A -85,B 0,C 180,E1 -32924.963,E2 -32924.963} C_VEL
LIN {X 0,Y 130.495,Z 597.2,A -85,B 0,C 180,E1 -32930.733,E2 -32930.733} C_VEL
LIN {X 0,Y 127.455,Z 589.021,A -85,B 0,C 180,E1 -32937.638,E2 -32937.638} C_VEL
LIN {X 0,Y 126.346,Z 580.554,A -85,B 0,C 180,E1 -32943.616,E2 -32943.616} C_VEL
LIN {X 0,Y 126.208,Z 573.278,A -85,B 0,C 180,E1 -32947.975,E2 -32947.975} C_VEL
LIN {X 0,Y 126.267,Z 565.238,A -85,B 0,C 180,E1 -32952.007,E2 -32952.007} C_VEL
LIN {X 0,Y 126.399,Z 555.545,A -85,B 0,C 180,E1 -32956.086,E2 -32956.086} C_VEL
LIN {X 0,Y 126.846,Z 542.684,A -85,B 0,C 180,E1 -32960.515,E2 -32960.515} C_VEL
LIN {X 0,Y 127.544,Z 528.885,A -85,B 0,C 180,E1 -32964.323,E2 -32964.323} C_VEL
LIN {X 0,Y 128.475,Z 514.913,A -85,B 0,C 180,E1 -32967.388,E2 -32967.388} C_VEL
LIN {X 0,Y 129.302,Z 501.516,A -85,B 0,C 180,E1 -32969.671,E2 -32969.671} C_VEL
LIN {X 0,Y 130.24,Z 487.03,A -85,B 0,C 180,E1 -32971.543,E2 -32971.543} C_VEL
LIN {X 0,Y 131.357,Z 460.726,A -85,B 0,C 180,E1 -32974.164,E2 -32974.164} C_VEL
LIN {X 0,Y 134.775,Z 394.623,A -85,B 0,C 180,E1 -32980.438,E2 -32980.438} C_VEL
LIN {X 0,Y 134.722,Z 394.03,A -85,B 0,C 180,E1 -32980.534,E2 -32980.534} C_VEL
LIN {X 0,Y 135.334,Z 398.001,A -85,B 0,C 180,E1 -32981.292,E2 -32981.292} C_VEL
LIN {X 0,Y 135.798,Z 398.396,A -85,B 0,C 180,E1 -32981.613,E2 -32981.613} C_VEL
LIN {X 0,Y 136.725,Z 397.821,A -85,B 0,C 180,E1 -32982.118,E2 -32982.118} C_VEL
LIN {X 0,Y 139.059,Z 394.015,A -85,B 0,C 180,E1 -32983.128,E2 -32983.128} C_VEL
LIN {X 0,Y 141.289,Z 388.042,A -85,B 0,C 180,E1 -32983.847,E2 -32983.847} C_VEL
LIN {X 0,Y 142.303,Z 384.741,A -85,B 0,C 180,E1 -32984.114,E2 -32984.114} C_VEL
LIN {X 0,Y 144.435,Z 383.577,A -85,B 0,C 180,E1 -32985.121,E2 -32985.121} C_VEL
LIN {X 0,Y 146.712,Z 380.768,A -85,B 0,C 180,E1 -32986.02,E2 -32986.02} C_VEL
LIN {X 0,Y 149.853,Z 374.687,A -85,B 0,C 180,E1 -32987.027,E2 -32987.027} C_VEL
LIN {X 0,Y 150.278,Z 374.846,A -85,B 0,C 180,E1 -32987.231,E2 -32987.231} C_VEL
LIN {X 0,Y 155.802,Z 384.637,A -85,B 0,C 180,E1 -32990.221,E2 -32990.221} C_VEL
LIN {X 0,Y 160.869,Z 395.141,A -85,B 0,C 180,E1 -32992.75,E2 -32992.75} C_VEL
LIN {X 0,Y 162.732,Z 399.36,A -85,B 0,C 180,E1 -32993.638,E2 -32993.638} C_VEL
LIN {X 0,Y 158.377,Z 461.472,A -85,B 0,C 180,E1 -32996.051,E2 -32996.051} C_VEL
LIN {X 0,Y 156.547,Z 475.691,A -85,B 0,C 180,E1 -32997.043,E2 -32997.043} C_VEL
LIN {X 0,Y 154.093,Z 489.398,A -85,B 0,C 180,E1 -32998.477,E2 -32998.477} C_VEL
LIN {X 0,Y 150.706,Z 503.151,A -85,B 0,C 180,E1 -33000.401,E2 -33000.401} C_VEL
LIN {X 0,Y 146.842,Z 515.54,A -85,B 0,C 180,E1 -33002.663,E2 -33002.663} C_VEL
LIN {X 0,Y 142.953,Z 526.83,A -85,B 0,C 180,E1 -33005.38,E2 -33005.38} C_VEL
LIN {X 0,Y 139.828,Z 535.256,A -85,B 0,C 180,E1 -33007.925,E2 -33007.925} C_VEL
LIN {X 0,Y 135.368,Z 545.947,A -85,B 0,C 180,E1 -33011.906,E2 -33011.906} C_VEL
LIN {X 0,Y 131.62,Z 554.763,A -85,B 0,C 180,E1 -33016.137,E2 -33016.137} C_VEL
LIN {X 0,Y 128.556,Z 562.099,A -85,B 0,C 180,E1 -33020.585,E2 -33020.585} C_VEL
LIN {X 0,Y 126.367,Z 568.196,A -85,B 0,C 180,E1 -33025.221,E2 -33025.221} C_VEL
LIN {X 0,Y 124.618,Z 573.289,A -85,B 0,C 180,E1 -33029.992,E2 -33029.992} C_VEL
LIN {X 0,Y 123.084,Z 578.576,A -85,B 0,C 180,E1 -33036.527,E2 -33036.527} C_VEL
LIN {X 0,Y 122.966,Z 582.341,A -85,B 0,C 180,E1 -33043.162,E2 -33043.162} C_VEL
LIN {X 0,Y 123.908,Z 584.718,A -85,B 0,C 180,E1 -33049.818,E2 -33049.818} C_VEL
LIN {X 0,Y 126.295,Z 585.723,A -85,B 0,C 180,E1 -33056.33,E2 -33056.33} C_VEL
LIN {X 0,Y 130.023,Z 585.369,A -85,B 0,C 180,E1 -33062.586,E2 -33062.586} C_VEL
LIN {X 0,Y 135.068,Z 583.638,A -85,B 0,C 180,E1 -33068.474,E2 -33068.474} C_VEL
LIN {X 0,Y 141.347,Z 580.451,A -85,B 0,C 180,E1 -33073.919,E2 -33073.919} C_VEL
LIN {X 0,Y 148.75,Z 575.684,A -85,B 0,C 180,E1 -33078.876,E2 -33078.876} C_VEL
LIN {X 0,Y 154.943,Z 571.035,A -85,B 0,C 180,E1 -33082.278,E2 -33082.278} C_VEL
LIN {X 0,Y 162.971,Z 563.976,A -85,B 0,C 180,E1 -33086.032,E2 -33086.032} C_VEL
LIN {X 0,Y 171.135,Z 555.627,A -85,B 0,C 180,E1 -33089.249,E2 -33089.249} C_VEL
LIN {X 0,Y 178.725,Z 546.662,A -85,B 0,C 180,E1 -33091.816,E2 -33091.816} C_VEL
LIN {X 0,Y 185.344,Z 537.616,A -85,B 0,C 180,E1 -33093.824,E2 -33093.824} C_VEL
LIN {X 0,Y 192.669,Z 525.796,A -85,B 0,C 180,E1 -33095.865,E2 -33095.865} C_VEL
LIN {X 0,Y 199.014,Z 513.461,A -85,B 0,C 180,E1 -33097.486,E2 -33097.486} C_VEL
LIN {X 0,Y 203.927,Z 501.719,A -85,B 0,C 180,E1 -33098.683,E2 -33098.683} C_VEL
LIN {X 0,Y 207.808,Z 490.138,A -85,B 0,C 180,E1 -33099.613,E2 -33099.613} C_VEL
LIN {X 0,Y 211.449,Z 475.89,A -85,B 0,C 180,E1 -33100.471,E2 -33100.471} C_VEL
LIN {X 0,Y 213.851,Z 462.147,A -85,B 0,C 180,E1 -33101.021,E2 -33101.021} C_VEL
LIN {X 0,Y 215.478,Z 445.766,A -85,B 0,C 180,E1 -33101.482,E2 -33101.482} C_VEL
LIN {X 0,Y 211.917,Z 438.154,A -85,B 0,C 180,E1 -33104.36,E2 -33104.36} C_VEL
LIN {X 0,Y 208.277,Z 431.064,A -85,B 0,C 180,E1 -33107.793,E2 -33107.793} C_VEL
LIN {X 0,Y 205.78,Z 426.438,A -85,B 0,C 180,E1 -33110.672,E2 -33110.672} C_VEL
LIN {X 0,Y 203.866,Z 422.929,A -85,B 0,C 180,E1 -33113.372,E2 -33113.372} C_VEL
LIN {X 0,Y 201.933,Z 419.131,A -85,B 0,C 180,E1 -33117.018,E2 -33117.018} C_VEL
LIN {X 0,Y 200.357,Z 415.822,A -85,B 0,C 180,E1 -33122.313,E2 -33122.313} C_VEL
LIN {X 0,Y 200.276,Z 415.105,A -85,B 0,C 180,E1 -33123.245,E2 -33123.245} C_VEL
LIN {X 0,Y 200.156,Z 415.253,A -85,B 0,C 180,E1 -33127.162,E2 -33127.162} C_VEL
LIN {X 0,Y 200.975,Z 418.626,A -85,B 0,C 180,E1 -33132.071,E2 -33132.071} C_VEL
LIN {X 0,Y 202.285,Z 421.606,A -85,B 0,C 180,E1 -33135.379,E2 -33135.379} C_VEL
LIN {X 0,Y 204.43,Z 427.074,A -85,B 0,C 180,E1 -33139.205,E2 -33139.205} C_VEL
LIN {X 0,Y 206.269,Z 431.706,A -85,B 0,C 180,E1 -33141.743,E2 -33141.743} C_VEL
LIN {X 0,Y 208.221,Z 436.635,A -85,B 0,C 180,E1 -33144.004,E2 -33144.004} C_VEL
LIN {X 0,Y 211.133,Z 444.582,A -85,B 0,C 180,E1 -33146.938,E2 -33146.938} C_VEL
LIN {X 0,Y 213.958,Z 453.298,A -85,B 0,C 180,E1 -33149.478,E2 -33149.478} C_VEL
LIN {X 0,Y 214.629,Z 455.538,A -85,B 0,C 180,E1 -33150.049,E2 -33150.049} C_VEL
LIN {X 0,Y 212.378,Z 475.808,A -85,B 0,C 180,E1 -33150.586,E2 -33150.586} C_VEL
LIN {X 0,Y 209.377,Z 490.496,A -85,B 0,C 180,E1 -33151.141,E2 -33151.141} C_VEL
LIN {X 0,Y 205.266,Z 504.593,A -85,B 0,C 180,E1 -33151.926,E2 -33151.926} C_VEL
LIN {X 0,Y 200.107,Z 517.73,A -85,B 0,C 180,E1 -33152.862,E2 -33152.862} C_VEL
LIN {X 0,Y 194.341,Z 529.65,A -85,B 0,C 180,E1 -33154.018,E2 -33154.018} C_VEL
LIN {X 0,Y 187.375,Z 541.724,A -85,B 0,C 180,E1 -33155.615,E2 -33155.615} C_VEL
LIN {X 0,Y 180.546,Z 551.747,A -85,B 0,C 180,E1 -33157.325,E2 -33157.325} C_VEL
LIN {X 0,Y 172.742,Z 561.738,A -85,B 0,C 180,E1 -33159.618,E2 -33159.618} C_VEL
LIN {X 0,Y 164.126,Z 571.301,A -85,B 0,C 180,E1 -33162.603,E2 -33162.603} C_VEL
LIN {X 0,Y 156.559,Z 578.524,A -85,B 0,C 180,E1 -33165.612,E2 -33165.612} C_VEL
LIN {X 0,Y 149.489,Z 584.553,A -85,B 0,C 180,E1 -33169.015,E2 -33169.015} C_VEL
LIN {X 0,Y 141.749,Z 590.357,A -85,B 0,C 180,E1 -33173.641,E2 -33173.641} C_VEL
LIN {X 0,Y 135.149,Z 594.646,A -85,B 0,C 180,E1 -33178.792,E2 -33178.792} C_VEL
LIN {X 0,Y 129.907,Z 597.546,A -85,B 0,C 180,E1 -33184.456,E2 -33184.456} C_VEL
LIN {X 0,Y 126.027,Z 599.132,A -85,B 0,C 180,E1 -33190.529,E2 -33190.529} C_VEL
LIN {X 0,Y 123.641,Z 599.435,A -85,B 0,C 180,E1 -33196.911,E2 -33196.911} C_VEL
LIN {X 0,Y 122.85,Z 598.459,A -85,B 0,C 180,E1 -33203.46,E2 -33203.46} C_VEL
LIN {X 0,Y 123.744,Z 596.188,A -85,B 0,C 180,E1 -33210.008,E2 -33210.008} C_VEL
LIN {X 0,Y 124.996,Z 593.521,A -85,B 0,C 180,E1 -33214.83,E2 -33214.83} C_VEL
LIN {X 0,Y 127.582,Z 588.75,A -85,B 0,C 180,E1 -33221.086,E2 -33221.086} C_VEL
LIN {X 0,Y 128.52,Z 596.143,A -85,B 0,C 180,E1 -33227.45,E2 -33227.45} C_VEL
LIN {X 0,Y 131.429,Z 602.253,A -85,B 0,C 180,E1 -33233.568,E2 -33233.568} C_VEL
LIN {X 0,Y 135.951,Z 607.069,A -85,B 0,C 180,E1 -33239.143,E2 -33239.143} C_VEL
LIN {X 0,Y 140.551,Z 610.173,A -85,B 0,C 180,E1 -33243.251,E2 -33243.251} C_VEL
LIN {X 0,Y 147.856,Z 613.265,A -85,B 0,C 180,E1 -33248.022,E2 -33248.022} C_VEL
LIN {X 0,Y 156.492,Z 615.382,A -85,B 0,C 180,E1 -33252.182,E2 -33252.182} C_VEL
LIN {X 0,Y 165.844,Z 616.495,A -85,B 0,C 180,E1 -33255.897,E2 -33255.897} C_VEL
LIN {X 0,Y 172.968,Z 616.698,A -85,B 0,C 180,E1 -33258.097,E2 -33258.097} C_VEL
LIN {X 0,Y 174.13,Z 616.701,A -85,B 0,C 180,E1 -33258.79,E2 -33258.79} C_VEL
LIN {X 0,Y 174.138,Z 616.619,A -85,B 0,C 180,E1 -33259.899,E2 -33259.899} C_VEL
LIN {X 0,Y 172.51,Z 616.491,A -85,B 0,C 180,E1 -33261.347,E2 -33261.347} C_VEL
LIN {X 0,Y 170.396,Z 616.323,A -85,B 0,C 180,E1 -33262.41,E2 -33262.41} C_VEL
LIN {X 0,Y 163.751,Z 615.701,A -85,B 0,C 180,E1 -33264.852,E2 -33264.852} C_VEL
LIN {X 0,Y 156.765,Z 614.568,A -85,B 0,C 180,E1 -33267.278,E2 -33267.278} C_VEL
LIN {X 0,Y 146.616,Z 611.902,A -85,B 0,C 180,E1 -33271.462,E2 -33271.462} C_VEL
LIN {X 0,Y 137.424,Z 607.844,A -85,B 0,C 180,E1 -33276.572,E2 -33276.572} C_VEL
LIN {X 0,Y 129.748,Z 602.236,A -85,B 0,C 180,E1 -33282.727,E2 -33282.727} C_VEL
